C09109=1136.601,82.163,-54.023,-179.519,6.650,149.079
C09110=1136.606,81.914,-54.006,-179.522,6.649,149.080
C09111=1136.612,81.665,-53.989,-179.524,6.648,149.080
C09112=1136.617,81.416,-53.971,-179.527,6.646,149.081
C09113=1136.621,81.166,-53.954,-179.530,6.644,149.081
C09114=1136.626,80.916,-53.937,-179.532,6.643,149.082
C09115=1136.631,80.667,-53.920,-179.536,6.642,149.082
C09116=1136.636,80.418,-53.903,-179.538,6.641,149.083
C09117=1136.642,80.168,-53.886,-179.541,6.639,149.083
C09118=1136.646,79.919,-53.869,-179.543,6.637,149.084
C09119=1136.651,79.651,-53.850,-179.547,6.636,149.084
C09120=1136.656,79.383,-53.832,-179.549,6.634,149.085
C09121=1136.662,79.114,-53.813,-179.552,6.633,149.085
C09122=1136.668,78.846,-53.795,-179.555,6.632,149.086
C09123=1136.672,78.596,-53.778,-179.558,6.630,149.086
C09124=1136.677,78.347,-53.761,-179.560,6.629,149.087
C09125=1136.682,78.097,-53.744,-179.563,6.627,149.087
C09126=1136.687,77.847,-53.727,-179.566,6.626,149.088
C09127=1136.692,77.599,-53.710,-179.569,6.624,149.088
C09128=1136.697,77.349,-53.693,-179.571,6.624,149.089
C09129=1136.702,77.100,-53.676,-179.574,6.622,149.089
C09130=1136.706,76.850,-53.659,-179.577,6.621,149.090
C09131=1136.712,76.601,-53.642,-179.580,6.619,149.090
C09132=1136.716,76.352,-53.626,-179.582,6.618,149.091
C09133=1136.722,76.102,-53.609,-179.585,6.616,149.091
C09134=1136.727,75.853,-53.592,-179.587,6.615,149.091
C09135=1136.732,75.603,-53.575,-179.591,6.614,149.092
C09136=1136.736,75.354,-53.558,-179.593,6.613,149.093
C09137=1136.741,75.105,-53.540,-179.596,6.611,149.093
C09138=1136.746,74.856,-53.524,-179.598,6.609,149.093
C09139=1136.751,74.606,-53.507,-179.601,6.608,149.094
C09140=1136.756,74.357,-53.490,-179.604,6.607,149.095
C09141=1136.761,74.108,-53.474,-179.606,6.606,149.095
C09142=1136.766,73.858,-53.456,-179.609,6.604,149.095
C09143=1136.771,73.609,-53.440,-179.612,6.603,149.096
C09144=1136.775,73.359,-53.423,-179.615,6.602,149.096
C09145=1136.781,73.110,-53.406,-179.617,6.600,149.097
C09146=1136.786,72.860,-53.390,-179.620,6.598,149.097
C09147=1136.790,72.610,-53.374,-179.623,6.597,149.098
C09148=1136.796,72.361,-53.357,-179.625,6.596,149.098
C09149=1136.801,72.112,-53.340,-179.628,6.595,149.099
C09150=1136.806,71.863,-53.324,-179.631,6.593,149.099
C09151=1136.811,71.613,-53.307,-179.633,6.592,149.100
C09152=1136.816,71.364,-53.290,-179.636,6.591,149.100
C09153=1136.821,71.115,-53.274,-179.639,6.589,149.101
C09154=1136.826,70.865,-53.256,-179.642,6.588,149.101
C09155=1136.830,70.616,-53.240,-179.644,6.587,149.102
C09156=1136.836,70.366,-53.224,-179.647,6.585,149.102
C09157=1136.840,70.117,-53.207,-179.650,6.584,149.103
C09158=1136.845,69.867,-53.190,-179.652,6.583,149.103
C09159=1136.850,69.618,-53.174,-179.655,6.581,149.104
C09160=1136.855,69.369,-53.157,-179.658,6.580,149.104
C09161=1136.860,69.120,-53.141,-179.661,6.578,149.105
C09162=1136.866,68.870,-53.124,-179.663,6.578,149.105
C09163=1136.870,68.620,-53.108,-179.666,6.576,149.106
C09164=1136.875,68.371,-53.091,-179.669,6.575,149.106
C09165=1136.880,68.122,-53.075,-179.671,6.574,149.107
C09166=1136.886,67.872,-53.058,-179.674,6.572,149.107
C09167=1136.890,67.623,-53.042,-179.677,6.570,149.108
C09168=1136.895,67.374,-53.025,-179.679,6.570,149.108
C09169=1136.900,67.124,-53.009,-179.682,6.568,149.109
C09170=1136.905,66.874,-52.993,-179.685,6.567,149.109
C09171=1136.910,66.626,-52.977,-179.687,6.566,149.110
C09172=1136.915,66.376,-52.959,-179.690,6.565,149.110
C09173=1136.920,66.126,-52.944,-179.693,6.563,149.111
C09174=1136.925,65.877,-52.927,-179.695,6.562,149.111
C09175=1136.930,65.628,-52.911,-179.698,6.561,149.112
C09176=1136.935,65.378,-52.895,-179.701,6.559,149.112
C09177=1136.940,65.129,-52.878,-179.704,6.558,149.113
C09178=1136.944,64.880,-52.862,-179.706,6.557,149.113
C09179=1136.950,64.630,-52.846,-179.709,6.555,149.114
C09180=1136.955,64.380,-52.829,-179.712,6.554,149.114
C09181=1136.960,64.132,-52.813,-179.714,6.553,149.115
C09182=1136.965,63.882,-52.797,-179.717,6.551,149.115
C09183=1136.970,63.633,-52.780,-179.719,6.551,149.116
C09184=1136.974,63.383,-52.764,-179.722,6.549,149.116
C09185=1136.980,63.134,-52.748,-179.725,6.548,149.117
C09186=1136.984,62.884,-52.732,-179.728,6.547,149.117
C09187=1136.989,62.635,-52.716,-179.730,6.545,149.118
C09188=1136.994,62.385,-52.700,-179.733,6.544,149.118
C09189=1136.999,62.136,-52.684,-179.735,6.543,149.119
C09190=1137.004,61.886,-52.668,-179.738,6.542,149.119
C09191=1137.009,61.637,-52.651,-179.741,6.540,149.120
C09192=1137.015,61.387,-52.635,-179.743,6.539,149.120
C09193=1137.020,61.138,-52.618,-179.746,6.538,149.120
C09194=1137.025,60.888,-52.603,-179.749,6.536,149.121
C09195=1137.030,60.639,-52.586,-179.752,6.535,149.122
C09196=1137.034,60.389,-52.570,-179.754,6.534,149.122
C09197=1137.040,60.140,-52.554,-179.758,6.532,149.123
C09198=1137.045,59.891,-52.538,-179.760,6.532,149.123
C09199=1137.049,59.641,-52.522,-179.762,6.530,149.124
C09200=1137.055,59.392,-52.506,-179.765,6.529,149.124
C09201=1137.059,59.142,-52.491,-179.768,6.528,149.125
C09202=1137.064,58.893,-52.474,-179.771,6.526,149.125
C09203=1137.069,58.644,-52.459,-179.773,6.525,149.126
C09204=1137.074,58.395,-52.442,-179.776,6.524,149.126
C09205=1137.079,58.145,-52.427,-179.779,6.522,149.127
C09206=1137.084,57.895,-52.411,-179.781,6.522,149.127
C09207=1137.089,57.646,-52.394,-179.784,6.520,149.128
C09208=1137.094,57.397,-52.379,-179.786,6.520,149.128
C09209=1137.099,57.147,-52.363,-179.789,6.518,149.129
C09210=1137.104,56.898,-52.347,-179.792,6.516,149.129
C09211=1137.109,56.648,-52.331,-179.794,6.516,149.130
C09212=1137.114,56.398,-52.315,-179.797,6.514,149.130
C09213=1137.120,56.149,-52.299,-179.799,6.513,149.131
C09214=1137.124,55.900,-52.283,-179.802,6.512,149.131
C09215=1137.129,55.650,-52.268,-179.805,6.510,149.132
C09216=1137.134,55.401,-52.252,-179.807,6.510,149.132
C09217=1137.139,55.151,-52.236,-179.810,6.508,149.133
C09218=1137.144,54.902,-52.220,-179.813,6.507,149.133
C09219=1137.150,54.653,-52.204,-179.816,6.506,149.134
C09220=1137.154,54.403,-52.188,-179.818,6.504,149.134
C09221=1137.159,54.154,-52.173,-179.821,6.504,149.135
C09222=1137.164,53.904,-52.158,-179.824,6.502,149.135
C09223=1137.170,53.636,-52.141,-179.827,6.500,149.136
C09224=1137.175,53.367,-52.123,-179.829,6.500,149.136
C09225=1137.180,53.098,-52.106,-179.832,6.498,149.137
C09226=1137.186,52.830,-52.089,-179.835,6.497,149.138
C09227=1137.191,52.580,-52.074,-179.837,6.496,149.138
C09228=1137.196,52.331,-52.059,-179.840,6.495,149.138
C09229=1137.201,52.081,-52.043,-179.843,6.493,149.139
C09230=1137.206,51.832,-52.027,-179.845,6.492,149.140
C09231=1137.211,51.583,-52.011,-179.848,6.491,149.140
C09232=1137.215,51.333,-51.996,-179.851,6.490,149.141
C09233=1137.221,51.084,-51.980,-179.854,6.489,149.141
C09234=1137.226,50.834,-51.964,-179.856,6.488,149.142
C09235=1137.232,50.585,-51.949,-179.859,6.487,149.142
C09236=1137.236,50.335,-51.933,-179.862,6.485,149.143
C09237=1137.241,50.086,-51.918,-179.864,6.484,149.143
C09238=1137.246,49.836,-51.902,-179.867,6.483,149.144
C09239=1137.252,49.587,-51.887,-179.869,6.482,149.144
C09240=1137.256,49.337,-51.871,-179.872,6.480,149.145
C09241=1137.261,49.088,-51.856,-179.874,6.480,149.145
C09242=1137.267,48.838,-51.840,-179.878,6.478,149.146
C09243=1137.271,48.589,-51.825,-179.880,6.477,149.146
C09244=1137.276,48.339,-51.809,-179.882,6.476,149.147
C09245=1137.281,48.090,-51.794,-179.886,6.475,149.147
C09246=1137.286,47.840,-51.779,-179.888,6.474,149.148
C09247=1137.291,47.591,-51.763,-179.891,6.472,149.148
C09248=1137.297,47.342,-51.747,-179.893,6.472,149.149
C09249=1137.301,47.092,-51.732,-179.896,6.470,149.149
C09250=1137.306,46.842,-51.716,-179.898,6.469,149.150
C09251=1137.311,46.593,-51.701,-179.901,6.468,149.150
C09252=1137.317,46.343,-51.687,-179.904,6.467,149.151
C09253=1137.322,46.094,-51.671,-179.906,6.466,149.151
C09254=1137.326,45.844,-51.656,-179.908,6.465,149.152
C09255=1137.331,45.595,-51.640,-179.912,6.463,149.152
C09256=1137.336,45.346,-51.625,-179.914,6.463,149.153
C09257=1137.341,45.096,-51.609,-179.917,6.461,149.153
C09258=1137.347,44.847,-51.594,-179.920,6.460,149.154
C09259=1137.352,44.597,-51.580,-179.922,6.459,149.154
C09260=1137.357,44.347,-51.564,-179.925,6.457,149.155
C09261=1137.361,44.098,-51.549,-179.927,6.457,149.156
C09262=1137.367,43.849,-51.533,-179.930,6.455,149.156
C09263=1137.371,43.599,-51.518,-179.932,6.454,149.156
C09264=1137.377,43.349,-51.503,-179.936,6.453,149.157
C09265=1137.382,43.100,-51.488,-179.938,6.452,149.158
C09266=1137.387,42.851,-51.473,-179.941,6.451,149.158
C09267=1137.392,42.602,-51.458,-179.943,6.450,149.159
C09268=1137.397,42.351,-51.442,-179.946,6.449,149.159
C09269=1137.401,42.102,-51.427,-179.948,6.448,149.160
C09270=1137.407,41.853,-51.412,-179.951,6.446,149.160
C09271=1137.411,41.604,-51.397,-179.954,6.446,149.161
C09272=1137.417,41.354,-51.382,-179.956,6.444,149.161
C09273=1137.422,41.104,-51.367,-179.959,6.444,149.162
C09274=1137.427,40.855,-51.351,-179.962,6.442,149.162
C09275=1137.432,40.605,-51.337,-179.964,6.441,149.163
C09276=1137.437,40.356,-51.322,-179.967,6.440,149.163
C09277=1137.442,40.107,-51.307,-179.969,6.439,149.164
C09278=1137.448,39.857,-51.292,-179.972,6.437,149.164
C09279=1137.452,39.608,-51.277,-179.975,6.437,149.165
C09280=1137.457,39.358,-51.261,-179.977,6.435,149.165
C09281=1137.462,39.108,-51.246,-179.980,6.434,149.166
C09282=1137.467,38.859,-51.231,-179.983,6.433,149.167
C09283=1137.473,38.609,-51.217,-179.985,6.432,149.167
C09284=1137.477,38.360,-51.202,-179.987,6.432,149.167
C09285=1137.483,38.110,-51.186,-179.990,6.430,149.168
C09286=1137.488,37.861,-51.172,-179.993,6.429,149.169
C09287=1137.493,37.611,-51.156,-179.995,6.428,149.169
C09288=1137.498,37.361,-51.142,-179.998,6.427,149.170
C09289=1137.503,37.112,-51.127,179.999,6.426,149.170
C09290=1137.508,36.862,-51.112,179.997,6.425,149.171
C09291=1137.513,36.613,-51.097,179.994,6.424,149.171
C09292=1137.518,36.364,-51.083,179.992,6.423,149.172
C09293=1137.523,36.114,-51.067,179.989,6.421,149.172
C09294=1137.528,35.864,-51.053,179.986,6.421,149.173
C09295=1137.533,35.615,-51.038,179.984,6.419,149.173
C09296=1137.539,35.365,-51.023,179.981,6.418,149.174
C09297=1137.543,35.116,-51.008,179.978,6.417,149.174
C09298=1137.548,34.867,-50.994,179.976,6.416,149.175
C09299=1137.554,34.617,-50.978,179.974,6.415,149.175
C09300=1137.558,34.367,-50.964,179.971,6.414,149.176
C09301=1137.563,34.118,-50.949,179.968,6.413,149.176
C09302=1137.569,33.868,-50.934,179.966,6.412,149.177
C09303=1137.574,33.619,-50.920,179.963,6.411,149.178
C09304=1137.578,33.370,-50.905,179.960,6.410,149.178
C09305=1137.584,33.121,-50.891,179.958,6.409,149.178
C09306=1137.589,32.871,-50.875,179.955,6.408,149.179
C09307=1137.594,32.621,-50.861,179.953,6.407,149.180
C09308=1137.599,32.372,-50.847,179.950,6.406,149.180
C09309=1137.604,32.123,-50.832,179.947,6.405,149.181
C09310=1137.610,31.873,-50.817,179.945,6.404,149.181
C09311=1137.615,31.623,-50.803,179.942,6.403,149.182
C09312=1137.619,31.374,-50.788,179.940,6.402,149.182
C09313=1137.624,31.124,-50.773,179.937,6.400,149.183
C09314=1137.630,30.874,-50.758,179.934,6.400,149.183
C09315=1137.635,30.625,-50.743,179.932,6.399,149.184
C09316=1137.639,30.375,-50.729,179.929,6.397,149.184
C09317=1137.644,30.126,-50.715,179.927,6.397,149.185
C09318=1137.650,29.877,-50.701,179.924,6.395,149.185
C09319=1137.655,29.627,-50.686,179.922,6.394,149.186
C09320=1137.660,29.377,-50.671,179.919,6.394,149.187
C09321=1137.665,29.128,-50.657,179.916,6.392,149.187
C09322=1137.670,28.878,-50.642,179.914,6.391,149.188
C09323=1137.675,28.629,-50.628,179.911,6.390,149.188
C09324=1137.680,28.379,-50.613,179.909,6.389,149.189
C09325=1137.685,28.129,-50.599,179.907,6.389,149.189
C09326=1137.691,27.880,-50.584,179.903,6.387,149.190
C09327=1137.696,27.611,-50.569,179.901,6.387,149.190
C09328=1137.701,27.343,-50.553,179.898,6.385,149.191
C09329=1137.707,27.073,-50.538,179.895,6.384,149.191
C09330=1137.712,26.804,-50.522,179.892,6.383,149.192
C09331=1137.718,26.554,-50.507,179.890,6.382,149.193
C09332=1137.723,26.305,-50.493,179.887,6.381,149.193
C09333=1137.728,26.056,-50.479,179.885,6.380,149.194
C09334=1137.733,25.806,-50.465,179.882,6.379,149.194
C09335=1137.738,25.556,-50.451,179.879,6.378,149.195
C09336=1137.743,25.307,-50.436,179.877,6.377,149.195
C09337=1137.748,25.057,-50.421,179.875,6.376,149.196
C09338=1137.753,24.808,-50.408,179.872,6.375,149.196
C09339=1137.758,24.559,-50.393,179.869,6.374,149.197
C09340=1137.763,24.309,-50.379,179.867,6.373,149.197
C09341=1137.768,24.059,-50.365,179.864,6.373,149.198
C09342=1137.773,23.810,-50.350,179.862,6.371,149.198
C09343=1137.779,23.561,-50.337,179.859,6.370,149.199
C09344=1137.783,23.311,-50.322,179.856,6.369,149.200
C09345=1137.788,23.061,-50.308,179.854,6.368,149.200
C09346=1137.793,22.811,-50.294,179.851,6.368,149.201
C09347=1137.798,22.562,-50.279,179.849,6.366,149.201
C09348=1137.804,22.313,-50.265,179.846,6.365,149.202
C09349=1137.809,22.063,-50.251,179.844,6.365,149.202
C09350=1137.814,21.813,-50.237,179.841,6.363,149.203
C09351=1137.819,21.564,-50.223,179.839,6.362,149.203
C09352=1137.824,21.315,-50.209,179.836,6.362,149.204
C09353=1137.829,21.065,-50.194,179.833,6.360,149.204
C09354=1137.834,20.815,-50.180,179.831,6.359,149.205
C09355=1137.839,20.565,-50.166,179.828,6.358,149.205
C09356=1137.845,20.316,-50.152,179.826,6.357,149.206
C09357=1137.850,20.067,-50.138,179.823,6.357,149.207
C09358=1137.855,19.816,-50.124,179.820,6.355,149.207
C09359=1137.861,19.567,-50.110,179.818,6.354,149.208
C09360=1137.865,19.318,-50.097,179.816,6.354,149.208
C09361=1137.870,19.068,-50.082,179.813,6.352,149.209
C09362=1137.875,18.819,-50.068,179.811,6.352,149.209
C09363=1137.880,18.570,-50.054,179.808,6.351,149.210
C09364=1137.885,18.320,-50.040,179.805,6.350,149.210
C09365=1137.890,18.069,-50.026,179.803,6.349,149.211
C09366=1137.896,17.820,-50.012,179.800,6.348,149.211
C09367=1137.901,17.571,-49.998,179.798,6.347,149.212
C09368=1137.906,17.321,-49.984,179.795,6.346,149.213
C09369=1137.911,17.072,-49.970,179.793,6.345,149.213
C09370=1137.916,16.823,-49.956,179.790,6.344,149.213
C09371=1137.921,16.572,-49.943,179.787,6.343,149.214
C09372=1137.926,16.323,-49.929,179.785,6.343,149.215
C09373=1137.931,16.074,-49.914,179.782,6.341,149.215
C09374=1137.936,15.824,-49.900,179.780,6.341,149.216
C09375=1137.942,15.575,-49.888,179.778,6.340,149.216
C09376=1137.946,15.325,-49.873,179.775,6.338,149.217
C09377=1137.951,15.075,-49.859,179.772,6.338,149.217
C09378=1137.957,14.826,-49.845,179.770,6.337,149.218
C09379=1137.962,14.576,-49.832,179.767,6.336,149.219
C09380=1137.967,14.327,-49.818,179.765,6.335,149.219
C09381=1137.972,14.077,-49.804,179.762,6.334,149.219
C09382=1137.977,13.827,-49.790,179.760,6.334,149.220
C09383=1137.983,13.578,-49.776,179.757,6.332,149.221
C09384=1137.987,13.329,-49.763,179.755,6.331,149.221
C09385=1137.992,13.078,-49.749,179.752,6.331,149.222
C09386=1137.998,12.829,-49.735,179.749,6.329,149.222
C09387=1138.003,12.580,-49.721,179.747,6.328,149.223
C09388=1138.008,12.330,-49.708,179.744,6.328,149.223
C09389=1138.013,12.081,-49.694,179.742,6.327,149.224
C09390=1138.019,11.831,-49.681,179.739,6.326,149.224
C09391=1138.024,11.581,-49.667,179.737,6.325,149.225
C09392=1138.028,11.332,-49.653,179.735,6.324,149.225
C09393=1138.034,11.082,-49.640,179.731,6.323,149.226
C09394=1138.039,10.833,-49.626,179.729,6.322,149.227
C09395=1138.044,10.583,-49.613,179.727,6.321,149.227
C09396=1138.049,10.333,-49.599,179.724,6.321,149.228
C09397=1138.055,10.084,-49.585,179.722,6.319,149.228
C09398=1138.059,9.834,-49.572,179.719,6.319,149.229
C09399=1138.064,9.585,-49.558,179.717,6.318,149.229
C09400=1138.070,9.335,-49.544,179.714,6.316,149.230
C09401=1138.074,9.086,-49.531,179.711,6.316,149.230
C09402=1138.080,8.836,-49.517,179.709,6.315,149.231
C09403=1138.085,8.586,-49.503,179.707,6.314,149.231
C09404=1138.090,8.337,-49.491,179.704,6.313,149.232
C09405=1138.095,8.087,-49.476,179.702,6.312,149.233
C09406=1138.101,7.838,-49.463,179.699,6.312,149.233
C09407=1138.105,7.588,-49.450,179.697,6.311,149.234
C09408=1138.111,7.339,-49.436,179.694,6.310,149.234
C09409=1138.115,7.089,-49.423,179.691,6.309,149.235
C09410=1138.121,6.840,-49.409,179.689,6.308,149.235
C09411=1138.126,6.589,-49.396,179.686,6.307,149.236
C09412=1138.131,6.341,-49.382,179.684,6.306,149.236
C09413=1138.136,6.090,-49.369,179.682,6.305,149.237
C09414=1138.141,5.841,-49.356,179.679,6.305,149.237
C09415=1138.146,5.591,-49.342,179.676,6.303,149.238
C09416=1138.151,5.342,-49.329,179.674,6.303,149.238
C09417=1138.156,5.092,-49.315,179.671,6.302,149.239
C09418=1138.161,4.843,-49.303,179.669,6.301,149.240
C09419=1138.167,4.593,-49.289,179.666,6.300,149.240
C09420=1138.172,4.344,-49.275,179.664,6.299,149.241
C09421=1138.177,4.094,-49.262,179.662,6.299,149.241
C09422=1138.183,3.844,-49.249,179.659,6.298,149.242
C09423=1138.187,3.595,-49.236,179.657,6.297,149.242
C09424=1138.193,3.345,-49.222,179.654,6.296,149.243
C09425=1138.198,3.096,-49.209,179.651,6.295,149.244
C09426=1138.203,2.846,-49.195,179.649,6.294,149.244
C09427=1138.208,2.597,-49.183,179.647,6.294,149.244
C09428=1138.213,2.346,-49.169,179.644,6.292,149.245
C09429=1138.218,2.097,-49.156,179.642,6.292,149.246
C09430=1138.224,1.848,-49.142,179.639,6.291,149.246
C09431=1138.229,1.578,-49.129,179.637,6.290,149.247
C09432=1138.235,1.308,-49.115,179.634,6.289,149.247
C09433=1138.240,1.039,-49.100,179.631,6.288,149.248
C09434=1138.246,0.770,-49.086,179.628,6.287,149.249
C09435=1138.251,0.519,-49.073,179.626,6.286,149.249
C09436=1138.256,0.271,-49.059,179.624,6.286,149.250
C09437=1138.261,0.021,-49.047,179.621,6.285,149.250
C09438=1138.266,-0.229,-49.033,179.618,6.283,149.251
C09439=1138.271,-0.478,-49.021,179.616,6.283,149.251
C09440=1138.277,-0.729,-49.007,179.613,6.282,149.252
C09441=1138.281,-0.977,-48.994,179.611,6.281,149.252
C09442=1138.287,-1.227,-48.981,179.609,6.281,149.253
C09443=1138.292,-1.477,-48.968,179.606,6.279,149.254
C09444=1138.297,-1.726,-48.955,179.604,6.279,149.254
C09445=1138.303,-1.976,-48.942,179.601,6.278,149.255
C09446=1138.307,-2.226,-48.929,179.599,6.277,149.255
C09447=1138.312,-2.475,-48.916,179.597,6.277,149.256
C09448=1138.318,-2.725,-48.903,179.593,6.275,149.256
C09449=1138.323,-2.975,-48.890,179.591,6.275,149.257
C09450=1138.328,-3.224,-48.876,179.589,6.274,149.257
C09451=1138.333,-3.473,-48.863,179.586,6.273,149.258
C09452=1138.338,-3.723,-48.851,179.584,6.273,149.258
C09453=1138.344,-3.973,-48.837,179.581,6.271,149.259
C09454=1138.349,-4.222,-48.825,179.579,6.271,149.260
C09455=1138.353,-4.472,-48.812,179.577,6.270,149.260
C09456=1138.359,-4.722,-48.799,179.574,6.269,149.261
C09457=1138.364,-4.971,-48.786,179.572,6.269,149.261
C09458=1138.369,-5.221,-48.773,179.570,6.268,149.262
C09459=1138.374,-5.470,-48.760,179.566,6.267,149.262
C09460=1138.380,-5.720,-48.747,179.564,6.266,149.263
C09461=1138.385,-5.969,-48.735,179.561,6.265,149.263
C09462=1138.390,-6.219,-48.722,179.559,6.264,149.264
C09463=1138.395,-6.469,-48.708,179.557,6.264,149.264
C09464=1138.401,-6.718,-48.696,179.554,6.263,149.265
C09465=1138.405,-6.968,-48.683,179.552,6.262,149.266
C09466=1138.410,-7.218,-48.670,179.549,6.261,149.266
C09467=1138.416,-7.467,-48.657,179.547,6.260,149.267
C09468=1138.421,-7.717,-48.644,179.545,6.260,149.267
C09469=1138.426,-7.967,-48.632,179.542,6.259,149.268
C09470=1138.431,-8.217,-48.620,179.540,6.258,149.268
C09471=1138.436,-8.466,-48.607,179.537,6.257,149.269
C09472=1138.442,-8.716,-48.594,179.534,6.256,149.270
C09473=1138.447,-8.966,-48.581,179.532,6.256,149.270
C09474=1138.452,-9.215,-48.568,179.530,6.255,149.270
C09475=1138.457,-9.464,-48.556,179.527,6.254,149.271
C09476=1138.462,-9.714,-48.543,179.525,6.254,149.272
C09477=1138.467,-9.964,-48.530,179.522,6.252,149.272
C09478=1138.473,-10.214,-48.518,179.520,6.252,149.273
C09479=1138.478,-10.463,-48.505,179.518,6.251,149.273
C09480=1138.483,-10.712,-48.492,179.515,6.250,149.274
C09481=1138.488,-10.962,-48.480,179.513,6.250,149.274
C09482=1138.493,-11.212,-48.467,179.511,6.249,149.275
C09483=1138.498,-11.461,-48.454,179.508,6.248,149.276
C09484=1138.504,-11.711,-48.442,179.506,6.248,149.276
C09485=1138.509,-11.961,-48.429,179.503,6.246,149.276
C09486=1138.514,-12.210,-48.417,179.500,6.246,149.277
C09487=1138.519,-12.460,-48.404,179.498,6.245,149.278
C09488=1138.524,-12.710,-48.392,179.495,6.244,149.278
C09489=1138.529,-12.959,-48.379,179.493,6.244,149.279
C09490=1138.534,-13.209,-48.367,179.491,6.243,149.279
C09491=1138.540,-13.458,-48.353,179.488,6.242,149.280
C09492=1138.545,-13.709,-48.341,179.486,6.241,149.280
C09493=1138.550,-13.958,-48.328,179.483,6.240,149.281
C09494=1138.555,-14.207,-48.316,179.481,6.240,149.282
C09495=1138.560,-14.457,-48.303,179.479,6.239,149.282
C09496=1138.566,-14.707,-48.291,179.476,6.238,149.283
C09497=1138.571,-14.956,-48.279,179.474,6.238,149.283
C09498=1138.576,-15.205,-48.266,179.472,6.237,149.284
C09499=1138.581,-15.456,-48.254,179.469,6.236,149.284
C09500=1138.586,-15.705,-48.241,179.467,6.236,149.285
C09501=1138.591,-15.955,-48.229,179.464,6.234,149.285
C09502=1138.597,-16.205,-48.217,179.461,6.234,149.286
C09503=1138.602,-16.454,-48.204,179.459,6.233,149.287
C09504=1138.607,-16.703,-48.192,179.457,6.232,149.287
C09505=1138.612,-16.953,-48.180,179.454,6.232,149.288
C09506=1138.617,-17.202,-48.167,179.452,6.231,149.288
C09507=1138.622,-17.453,-48.155,179.449,6.230,149.289
C09508=1138.627,-17.702,-48.142,179.447,6.230,149.289
C09509=1138.632,-17.952,-48.130,179.445,6.229,149.290
C09510=1138.638,-18.202,-48.118,179.442,6.228,149.290
C09511=1138.643,-18.451,-48.105,179.440,6.227,149.291
C09512=1138.648,-18.701,-48.093,179.437,6.226,149.291
C09513=1138.654,-18.950,-48.081,179.435,6.226,149.292
C09514=1138.659,-19.200,-48.069,179.433,6.225,149.293
C09515=1138.664,-19.449,-48.056,179.430,6.224,149.293
C09516=1138.670,-19.699,-48.044,179.428,6.224,149.294
C09517=1138.675,-19.949,-48.032,179.426,6.223,149.294
C09518=1138.680,-20.199,-48.020,179.423,6.222,149.295
C09519=1138.685,-20.449,-48.007,179.421,6.222,149.295
C09520=1138.690,-20.699,-47.995,179.419,6.221,149.296
C09521=1138.695,-20.948,-47.982,179.416,6.220,149.297
C09522=1138.701,-21.198,-47.971,179.413,6.219,149.297
C09523=1138.706,-21.447,-47.958,179.411,6.218,149.298
C09524=1138.711,-21.697,-47.946,179.408,6.218,149.298
C09525=1138.716,-21.946,-47.933,179.406,6.217,149.299
C09526=1138.722,-22.196,-47.922,179.404,6.216,149.299
C09527=1138.726,-22.445,-47.910,179.401,6.216,149.300
C09528=1138.732,-22.695,-47.898,179.399,6.215,149.300
C09529=1138.737,-22.945,-47.885,179.397,6.214,149.301
C09530=1138.742,-23.195,-47.873,179.394,6.214,149.301
C09531=1138.748,-23.445,-47.861,179.392,6.213,149.302
C09532=1138.753,-23.694,-47.849,179.389,6.212,149.303
C09533=1138.758,-23.944,-47.837,179.387,6.212,149.303
C09534=1138.763,-24.193,-47.824,179.385,6.211,149.304
C09535=1138.769,-24.463,-47.812,179.382,6.210,149.304
C09536=1138.774,-24.733,-47.799,179.379,6.209,149.305
C09537=1138.780,-25.003,-47.786,179.377,6.208,149.305
C09538=1138.786,-25.273,-47.773,179.375,6.208,149.306
C09539=1138.791,-25.523,-47.761,179.372,6.207,149.307
C09540=1138.796,-25.772,-47.749,179.370,6.206,149.307
C09541=1138.802,-26.022,-47.737,179.368,6.206,149.308
C09542=1138.807,-26.272,-47.725,179.365,6.205,149.308
C09543=1138.811,-26.521,-47.713,179.363,6.204,149.309
C09544=1138.817,-26.771,-47.701,179.360,6.204,149.309
C09545=1138.822,-27.021,-47.689,179.357,6.202,149.310
C09546=1138.827,-27.270,-47.676,179.355,6.202,149.310
C09547=1138.832,-27.520,-47.665,179.352,6.201,149.311
C09548=1138.838,-27.770,-47.653,179.350,6.200,149.312
C09549=1138.843,-28.020,-47.641,179.348,6.200,149.312
C09550=1138.848,-28.269,-47.629,179.345,6.199,149.313
C09551=1138.853,-28.519,-47.617,179.343,6.198,149.313
C09552=1138.858,-28.769,-47.606,179.341,6.198,149.314
C09553=1138.864,-29.019,-47.594,179.338,6.197,149.314
C09554=1138.869,-29.268,-47.581,179.336,6.197,149.315
C09555=1138.873,-29.518,-47.570,179.334,6.196,149.315
C09556=1138.880,-29.767,-47.558,179.331,6.195,149.316
C09557=1138.885,-30.017,-47.546,179.329,6.195,149.316
C09558=1138.890,-30.267,-47.535,179.327,6.194,149.317
C09559=1138.895,-30.516,-47.523,179.324,6.193,149.318
C09560=1138.900,-30.766,-47.511,179.322,6.193,149.318
C09561=1138.906,-31.016,-47.499,179.319,6.192,149.319
C09562=1138.910,-31.265,-47.487,179.317,6.191,149.319
C09563=1138.916,-31.515,-47.476,179.315,6.191,149.320
C09564=1138.921,-31.765,-47.464,179.312,6.190,149.320
C09565=1138.926,-32.015,-47.452,179.310,6.189,149.321
C09566=1138.932,-32.263,-47.440,179.308,6.189,149.321
C09567=1138.937,-32.513,-47.428,179.305,6.188,149.322
C09568=1138.942,-32.763,-47.417,179.303,6.187,149.323
C09569=1138.947,-33.013,-47.405,179.301,6.187,149.323
C09570=1138.953,-33.263,-47.393,179.298,6.186,149.324
C09571=1138.957,-33.512,-47.382,179.296,6.185,149.324
C09572=1138.963,-33.762,-47.370,179.294,6.185,149.325
C09573=1138.969,-34.012,-47.359,179.291,6.184,149.325
C09574=1138.973,-34.261,-47.347,179.289,6.183,149.326
C09575=1138.979,-34.511,-47.335,179.287,6.183,149.326
C09576=1138.984,-34.761,-47.324,179.284,6.182,149.327
C09577=1138.989,-35.011,-47.312,179.282,6.182,149.328
C09578=1138.994,-35.261,-47.300,179.280,6.181,149.328
C09579=1139.000,-35.510,-47.289,179.277,6.180,149.329
C09580=1139.005,-35.760,-47.278,179.275,6.180,149.329
C09581=1139.010,-36.009,-47.266,179.273,6.179,149.330
C09582=1139.015,-36.259,-47.254,179.270,6.178,149.330
C09583=1139.021,-36.509,-47.242,179.268,6.178,149.331
C09584=1139.026,-36.758,-47.232,179.266,6.177,149.331
C09585=1139.031,-37.008,-47.220,179.263,6.176,149.332
C09586=1139.036,-37.258,-47.208,179.261,6.176,149.333
C09587=1139.041,-37.508,-47.196,179.259,6.175,149.333
C09588=1139.046,-37.757,-47.185,179.256,6.174,149.334
C09589=1139.052,-38.006,-47.174,179.254,6.174,149.334
C09590=1139.057,-38.256,-47.162,179.252,6.173,149.335
C09591=1139.062,-38.506,-47.150,179.249,6.172,149.335
C09592=1139.067,-38.756,-47.139,179.247,6.172,149.336
C09593=1139.072,-39.005,-47.127,179.245,6.171,149.336
C09594=1139.078,-39.254,-47.116,179.242,6.171,149.337
C09595=1139.083,-39.504,-47.104,179.240,6.170,149.337
C09596=1139.089,-39.755,-47.093,179.238,6.169,149.338
C09597=1139.094,-40.005,-47.082,179.236,6.169,149.339
C09598=1139.100,-40.254,-47.071,179.233,6.169,149.339
C09599=1139.104,-40.503,-47.059,179.231,6.168,149.340
C09600=1139.109,-40.753,-47.048,179.229,6.167,149.340
C09601=1139.114,-41.003,-47.036,179.226,6.167,149.341
C09602=1139.120,-41.252,-47.025,179.224,6.166,149.341
C09603=1139.125,-41.502,-47.014,179.222,6.165,149.342
C09604=1139.130,-41.752,-47.003,179.219,6.165,149.342
C09605=1139.136,-42.001,-46.991,179.217,6.164,149.343
C09606=1139.141,-42.251,-46.980,179.215,6.163,149.344
C09607=1139.146,-42.501,-46.968,179.212,6.163,149.344
C09608=1139.151,-42.750,-46.957,179.210,6.162,149.345
C09609=1139.157,-43.000,-46.946,179.207,6.162,149.345
C09610=1139.162,-43.250,-46.935,179.205,6.161,149.346
C09611=1139.167,-43.500,-46.923,179.203,6.160,149.346
C09612=1139.173,-43.749,-46.912,179.200,6.160,149.347
C09613=1139.178,-43.999,-46.901,179.198,6.159,149.347
C09614=1139.183,-44.249,-46.889,179.196,6.158,149.348
C09615=1139.188,-44.499,-46.878,179.193,6.158,149.349
C09616=1139.193,-44.748,-46.867,179.192,6.158,149.349
C09617=1139.199,-44.998,-46.856,179.190,6.157,149.350
C09618=1139.204,-45.248,-46.845,179.187,6.156,149.350
C09619=1139.209,-45.497,-46.834,179.185,6.156,149.351
C09620=1139.215,-45.747,-46.823,179.183,6.155,149.351
C09621=1139.219,-45.997,-46.811,179.180,6.155,149.352
C09622=1139.225,-46.246,-46.800,179.178,6.154,149.352
C09623=1139.230,-46.496,-46.789,179.176,6.153,149.353
C09624=1139.235,-46.746,-46.778,179.173,6.153,149.354
C09625=1139.241,-46.995,-46.766,179.171,6.152,149.354
C09626=1139.246,-47.245,-46.756,179.168,6.151,149.354
C09627=1139.251,-47.495,-46.744,179.166,6.151,149.355
C09628=1139.257,-47.744,-46.733,179.164,6.150,149.356
C09629=1139.262,-47.995,-46.722,179.162,6.150,149.356
C09630=1139.267,-48.243,-46.711,179.160,6.149,149.357
C09631=1139.273,-48.493,-46.700,179.157,6.149,149.357
C09632=1139.278,-48.744,-46.689,179.155,6.148,149.358
C09633=1139.283,-48.993,-46.678,179.153,6.147,149.358
C09634=1139.288,-49.243,-46.668,179.150,6.147,149.359
C09635=1139.293,-49.493,-46.656,179.148,6.146,149.359
C09636=1139.299,-49.742,-46.645,179.146,6.145,149.360
C09637=1139.304,-49.992,-46.634,179.143,6.145,149.361
C09638=1139.310,-50.241,-46.623,179.141,6.144,149.361
C09639=1139.314,-50.512,-46.611,179.139,6.143,149.362
C09640=1139.320,-50.783,-46.599,179.136,6.143,149.362
C09641=1139.327,-51.054,-46.588,179.134,6.142,149.363
C09642=1139.332,-51.325,-46.575,179.131,6.142,149.364
C09643=1139.337,-51.574,-46.564,179.129,6.141,149.364
C09644=1139.342,-51.824,-46.554,179.126,6.141,149.365
C09645=1139.347,-52.073,-46.542,179.124,6.140,149.365
C09646=1139.354,-52.323,-46.532,179.123,6.140,149.366
C09647=1139.358,-52.573,-46.520,179.120,6.139,149.366
C09648=1139.364,-52.822,-46.510,179.118,6.139,149.367
C09649=1139.368,-53.072,-46.499,179.116,6.138,149.367
C09650=1139.373,-53.322,-46.488,179.113,6.137,149.368
C09651=1139.380,-53.572,-46.477,179.111,6.137,149.368
C09652=1139.385,-53.822,-46.466,179.108,6.136,149.369
C09653=1139.390,-54.071,-46.455,179.106,6.135,149.369
C09654=1139.395,-54.321,-46.445,179.104,6.136,149.370
C09655=1139.400,-54.571,-46.435,179.102,6.135,149.371
C09656=1139.405,-54.820,-46.423,179.100,6.134,149.371
C09657=1139.411,-55.070,-46.412,179.097,6.134,149.372
C09658=1139.416,-55.320,-46.401,179.095,6.133,149.372
C09659=1139.422,-55.569,-46.391,179.093,6.132,149.373
C09660=1139.427,-55.819,-46.380,179.091,6.131,149.373
C09661=1139.431,-56.069,-46.369,179.088,6.131,149.374
C09662=1139.437,-56.319,-46.359,179.086,6.131,149.374
C09663=1139.442,-56.568,-46.348,179.084,6.130,149.375
C09664=1139.447,-56.818,-46.337,179.081,6.130,149.376
C09665=1139.453,-57.068,-46.326,179.079,6.129,149.376
C09666=1139.458,-57.317,-46.315,179.077,6.128,149.377
C09667=1139.463,-57.568,-46.305,179.075,6.127,149.377
C09668=1139.469,-57.817,-46.294,179.072,6.127,149.378
C09669=1139.474,-58.067,-46.283,179.071,6.127,149.378
C09670=1139.479,-58.316,-46.273,179.068,6.126,149.379
C09671=1139.484,-58.566,-46.262,179.066,6.126,149.379
C09672=1139.489,-58.815,-46.251,179.064,6.125,149.380
C09673=1139.494,-59.066,-46.241,179.061,6.124,149.380
C09674=1139.500,-59.315,-46.231,179.059,6.124,149.381
C09675=1139.505,-59.565,-46.219,179.057,6.123,149.382
C09676=1139.510,-59.814,-46.209,179.055,6.123,149.382
C09677=1139.517,-60.064,-46.198,179.053,6.122,149.383
C09678=1139.522,-60.314,-46.188,179.050,6.122,149.383
C09679=1139.527,-60.563,-46.177,179.048,6.121,149.384
C09680=1139.532,-60.814,-46.166,179.046,6.121,149.384
C09681=1139.538,-61.063,-46.156,179.044,6.120,149.385
C09682=1139.543,-61.313,-46.146,179.041,6.120,149.385
C09683=1139.548,-61.562,-46.135,179.039,6.119,149.386
C09684=1139.553,-61.813,-46.124,179.037,6.119,149.386
C09685=1139.558,-62.062,-46.114,179.034,6.118,149.387
C09686=1139.563,-62.312,-46.103,179.032,6.118,149.388
C09687=1139.569,-62.562,-46.093,179.030,6.117,149.388
C09688=1139.574,-62.811,-46.082,179.028,6.117,149.388
C09689=1139.579,-63.061,-46.072,179.026,6.116,149.389
C09690=1139.585,-63.311,-46.061,179.024,6.116,149.390
C09691=1139.590,-63.561,-46.051,179.021,6.115,149.390
C09692=1139.596,-63.810,-46.041,179.019,6.114,149.391
C09693=1139.601,-64.060,-46.030,179.017,6.114,149.391
C09694=1139.606,-64.310,-46.019,179.015,6.114,149.392
C09695=1139.611,-64.559,-46.009,179.013,6.113,149.392
C09696=1139.616,-64.809,-45.999,179.010,6.113,149.393
C09697=1139.621,-65.059,-45.989,179.008,6.112,149.393
C09698=1139.627,-65.308,-45.978,179.006,6.111,149.394
C09699=1139.632,-65.558,-45.968,179.003,6.110,149.394
C09700=1139.638,-65.808,-45.958,179.001,6.111,149.395
C09701=1139.643,-66.058,-45.947,178.999,6.110,149.396
C09702=1139.648,-66.308,-45.937,178.997,6.109,149.396
C09703=1139.653,-66.557,-45.926,178.995,6.108,149.397
C09704=1139.658,-66.807,-45.915,178.992,6.108,149.397
C09705=1139.664,-67.056,-45.905,178.991,6.108,149.398
C09706=1139.670,-67.306,-45.895,178.988,6.107,149.398
C09707=1139.675,-67.556,-45.884,178.986,6.107,149.399
C09708=1139.680,-67.806,-45.874,178.984,6.106,149.399
C09709=1139.685,-68.055,-45.865,178.981,6.105,149.400
C09710=1139.690,-68.305,-45.854,178.980,6.105,149.400
C09711=1139.696,-68.555,-45.844,178.977,6.105,149.401
C09712=1139.701,-68.804,-45.834,178.975,6.104,149.402
C09713=1139.706,-69.055,-45.823,178.973,6.103,149.402
C09714=1139.712,-69.304,-45.813,178.970,6.103,149.403
C09715=1139.717,-69.554,-45.803,178.968,6.103,149.403
C09716=1139.722,-69.804,-45.792,178.966,6.102,149.404
C09717=1139.727,-70.053,-45.782,178.964,6.102,149.404
C09718=1139.733,-70.303,-45.772,178.962,6.101,149.405
C09719=1139.738,-70.553,-45.762,178.959,6.100,149.405
C09720=1139.743,-70.802,-45.751,178.958,6.100,149.406
C09721=1139.749,-71.052,-45.741,178.955,6.100,149.406
C09722=1139.754,-71.302,-45.731,178.953,6.099,149.407
C09723=1139.759,-71.551,-45.721,178.951,6.099,149.408
C09724=1139.765,-71.801,-45.711,178.949,6.099,149.408
C09725=1139.770,-72.052,-45.701,178.947,6.098,149.409
C09726=1139.775,-72.301,-45.691,178.945,6.097,149.409
C09727=1139.781,-72.551,-45.681,178.942,6.097,149.410
C09728=1139.786,-72.800,-45.671,178.940,6.096,149.410
C09729=1139.791,-73.050,-45.660,178.938,6.096,149.411
C09730=1139.797,-73.300,-45.650,178.936,6.095,149.411
C09731=1139.802,-73.550,-45.640,178.933,6.095,149.412
C09732=1139.808,-73.799,-45.630,178.931,6.094,149.412
C09733=1139.812,-74.049,-45.620,178.929,6.094,149.413
C09734=1139.818,-74.299,-45.610,178.927,6.093,149.413
C09735=1139.823,-74.549,-45.600,178.925,6.093,149.414
C09736=1139.829,-74.798,-45.590,178.922,6.092,149.415
C09737=1139.833,-75.048,-45.580,178.921,6.092,149.415
C09738=1139.839,-75.298,-45.570,178.919,6.091,149.415
C09739=1139.845,-75.547,-45.559,178.916,6.091,149.416
C09740=1139.850,-75.797,-45.550,178.914,6.090,149.417
C09741=1139.855,-76.047,-45.540,178.912,6.090,149.417
C09742=1139.860,-76.297,-45.530,178.910,6.090,149.418
C09743=1139.866,-76.569,-45.518,178.907,6.089,149.418
C09744=1139.872,-76.840,-45.508,178.905,6.088,149.419
C09745=1139.877,-77.111,-45.497,178.903,6.088,149.419
C09746=1139.883,-77.383,-45.486,178.900,6.087,149.420
C09747=1139.889,-77.633,-45.476,178.898,6.087,149.421
C09748=1139.894,-77.882,-45.467,178.896,6.087,149.421
C09749=1139.900,-78.132,-45.457,178.894,6.086,149.422
C09750=1139.905,-78.381,-45.446,178.892,6.085,149.422
C09751=1139.910,-78.632,-45.437,178.889,6.085,149.423
C09752=1139.916,-78.881,-45.427,178.888,6.085,149.423
C09753=1139.921,-79.131,-45.417,178.886,6.084,149.424
C09754=1139.926,-79.381,-45.408,178.883,6.084,149.424
C09755=1139.932,-79.630,-45.398,178.881,6.083,149.425
C09756=1139.937,-79.880,-45.387,178.879,6.083,149.425
C09757=1139.942,-80.130,-45.377,178.877,6.082,149.426
C09758=1139.948,-80.380,-45.368,178.874,6.082,149.427
C09759=1139.953,-80.629,-45.358,178.873,6.082,149.427
C09760=1139.958,-80.879,-45.348,178.870,6.081,149.427
C09761=1139.964,-81.129,-45.339,178.868,6.080,149.428
C09762=1139.968,-81.379,-45.329,178.866,6.079,149.428
C09763=1139.974,-81.628,-45.318,178.864,6.080,149.429
C09764=1139.980,-81.878,-45.309,178.862,6.079,149.430
C09765=1139.985,-82.128,-45.299,178.860,6.078,149.430
C09766=1139.991,-82.378,-45.290,178.857,6.078,149.431
C09767=1139.995,-82.627,-45.280,178.856,6.078,149.431
C09768=1140.000,-82.877,-45.270,178.853,6.077,149.432
C09769=1140.006,-83.127,-45.260,178.851,6.076,149.432
C09770=1140.011,-83.377,-45.250,178.849,6.076,149.433
C09771=1140.017,-83.627,-45.241,178.847,6.076,149.433
C09772=1140.022,-83.876,-45.231,178.845,6.075,149.434
C09773=1140.028,-84.126,-45.221,178.842,6.075,149.434
C09774=1140.033,-84.375,-45.212,178.841,6.075,149.435
C09775=1140.038,-84.625,-45.202,178.839,6.074,149.435
C09776=1140.044,-84.876,-45.192,178.836,6.073,149.436
C09777=1140.048,-85.125,-45.183,178.835,6.073,149.436
C09778=1140.054,-85.375,-45.173,178.832,6.073,149.437
C09779=1140.059,-85.624,-45.163,178.830,6.072,149.438
C09780=1140.065,-85.874,-45.153,178.828,6.071,149.438
C09781=1140.070,-86.124,-45.144,178.826,6.071,149.439
C09782=1140.076,-86.373,-45.134,178.824,6.071,149.439
C09783=1140.081,-86.623,-45.125,178.821,6.070,149.440
C09784=1140.086,-86.873,-45.115,178.820,6.070,149.440
C09785=1140.091,-87.123,-45.106,178.817,6.069,149.441
C09786=1140.097,-87.373,-45.096,178.815,6.069,149.441
C09787=1140.102,-87.623,-45.087,178.814,6.069,149.442
C09788=1140.107,-87.872,-45.076,178.811,6.068,149.442
C09789=1140.112,-88.122,-45.068,178.809,6.068,149.443
C09790=1140.118,-88.372,-45.057,178.807,6.067,149.443
C09791=1140.123,-88.622,-45.048,178.805,6.067,149.444
C09792=1140.128,-88.871,-45.040,178.803,6.066,149.444
C09793=1140.134,-89.121,-45.029,178.801,6.065,149.445
C09794=1140.139,-89.371,-45.020,178.799,6.066,149.446
C09795=1140.145,-89.620,-45.010,178.796,6.065,149.446
C09796=1140.150,-89.870,-45.001,178.794,6.064,149.446
C09797=1140.156,-90.120,-44.991,178.793,6.064,149.447
C09798=1140.161,-90.370,-44.982,178.790,6.064,149.447
C09799=1140.167,-90.620,-44.973,178.788,6.063,149.448
C09800=1140.171,-90.869,-44.963,178.786,6.063,149.449
C09801=1140.177,-91.119,-44.954,178.784,6.062,149.449
C09802=1140.182,-91.369,-44.944,178.782,6.062,149.450
C09803=1140.187,-91.619,-44.935,178.780,6.062,149.450
C09804=1140.193,-91.869,-44.925,178.778,6.061,149.451
C09805=1140.198,-92.118,-44.916,178.775,6.061,149.451
C09806=1140.203,-92.368,-44.907,178.774,6.061,149.452
C09807=1140.209,-92.618,-44.897,178.771,6.060,149.452
C09808=1140.213,-92.868,-44.888,178.769,6.059,149.453
C09809=1140.219,-93.118,-44.878,178.768,6.059,149.453
C09810=1140.225,-93.368,-44.869,178.765,6.058,149.454
C09811=1140.229,-93.617,-44.860,178.763,6.058,149.454
C09812=1140.235,-93.867,-44.850,178.761,6.058,149.455
C09813=1140.240,-94.117,-44.841,178.759,6.057,149.455
C09814=1140.246,-94.366,-44.831,178.757,6.057,149.456
C09815=1140.251,-94.616,-44.822,178.755,6.057,149.456
C09816=1140.256,-94.866,-44.813,178.753,6.056,149.457
C09817=1140.262,-95.116,-44.803,178.751,6.055,149.457
C09818=1140.267,-95.365,-44.794,178.749,6.056,149.458
C09819=1140.272,-95.615,-44.785,178.747,6.055,149.459
C09820=1140.279,-95.865,-44.776,178.744,6.054,149.459
C09821=1140.284,-96.114,-44.767,178.743,6.054,149.460
C09822=1140.289,-96.364,-44.758,178.741,6.053,149.460
C09823=1140.295,-96.614,-44.748,178.738,6.053,149.460
C09824=1140.300,-96.864,-44.739,178.736,6.053,149.461
C09825=1140.305,-97.113,-44.730,178.734,6.052,149.462
C09826=1140.311,-97.363,-44.720,178.732,6.051,149.462
C09827=1140.316,-97.613,-44.711,178.730,6.051,149.463
C09828=1140.321,-97.863,-44.702,178.728,6.051,149.463
C09829=1140.326,-98.113,-44.693,178.726,6.050,149.464
C09830=1140.332,-98.362,-44.683,178.724,6.050,149.464
C09831=1140.337,-98.612,-44.674,178.722,6.050,149.465
C09832=1140.342,-98.862,-44.665,178.720,6.050,149.465
C09833=1140.348,-99.112,-44.656,178.718,6.049,149.466
C09834=1140.353,-99.362,-44.647,178.716,6.048,149.466
C09835=1140.358,-99.611,-44.637,178.714,6.048,149.467
C09836=1140.364,-99.860,-44.629,178.712,6.047,149.467
C09837=1140.370,-100.111,-44.619,178.710,6.047,149.468
C09838=1140.375,-100.360,-44.611,178.708,6.047,149.468
C09839=1140.380,-100.610,-44.602,178.705,6.046,149.469
C09840=1140.385,-100.860,-44.593,178.703,6.046,149.469
C09841=1140.391,-101.110,-44.583,178.702,6.046,149.470
C09842=1140.396,-101.360,-44.574,178.699,6.045,149.470
C09843=1140.401,-101.609,-44.565,178.698,6.045,149.471
C09844=1140.406,-101.859,-44.556,178.696,6.044,149.471
C09845=1140.412,-102.109,-44.547,178.693,6.043,149.472
C09846=1140.417,-102.359,-44.537,178.692,6.043,149.472
C09847=1140.424,-102.631,-44.528,178.689,6.043,149.473
C09848=1140.429,-102.903,-44.518,178.687,6.042,149.474
C09849=1140.435,-103.176,-44.509,178.685,6.042,149.474
C09850=1140.441,-103.448,-44.498,178.683,6.042,149.475
C09851=1140.446,-103.697,-44.489,178.680,6.041,149.475
C09852=1140.451,-103.947,-44.481,178.678,6.041,149.476
C09853=1140.457,-104.197,-44.471,178.677,6.041,149.476
C09854=1140.463,-104.447,-44.462,178.674,6.040,149.477
C09855=1140.468,-104.696,-44.454,178.673,6.040,149.477
C09856=1140.473,-104.946,-44.445,178.671,6.039,149.478
C09857=1140.478,-105.196,-44.436,178.668,6.039,149.478
C09858=1140.483,-105.446,-44.427,178.666,6.039,149.479
C09859=1140.488,-105.696,-44.418,178.664,6.038,149.479
C09860=1140.495,-105.945,-44.409,178.662,6.037,149.480
C09861=1140.500,-106.195,-44.400,178.660,6.037,149.480
C09862=1140.505,-106.445,-44.391,178.658,6.037,149.481
C09863=1140.510,-106.695,-44.382,178.657,6.037,149.481
C09864=1140.516,-106.945,-44.373,178.654,6.036,149.482
C09865=1140.521,-107.195,-44.364,178.652,6.035,149.482
C09866=1140.527,-107.444,-44.356,178.651,6.035,149.483
C09867=1140.532,-107.694,-44.347,178.648,6.035,149.483
C09868=1140.537,-107.943,-44.338,178.646,6.035,149.484
C09869=1140.543,-108.194,-44.329,178.644,6.034,149.484
C09870=1140.548,-108.443,-44.320,178.643,6.034,149.485
C09871=1140.553,-108.693,-44.311,178.640,6.033,149.485
C09872=1140.559,-108.943,-44.303,178.638,6.033,149.486
C09873=1140.564,-109.193,-44.294,178.637,6.033,149.486
C09874=1140.570,-109.443,-44.285,178.634,6.032,149.487
C09875=1140.575,-109.693,-44.276,178.633,6.032,149.487
C09876=1140.580,-109.942,-44.267,178.631,6.031,149.488
C09877=1140.586,-110.192,-44.259,178.628,6.031,149.488
C09878=1140.591,-110.441,-44.250,178.627,6.031,149.489
C09879=1140.596,-110.691,-44.241,178.624,6.030,149.490
C09880=1140.601,-110.941,-44.232,178.623,6.030,149.490
C09881=1140.607,-111.191,-44.224,178.620,6.030,149.490
C09882=1140.612,-111.441,-44.215,178.618,6.029,149.491
C09883=1140.618,-111.691,-44.207,178.617,6.029,149.491
C09884=1140.623,-111.940,-44.198,178.614,6.028,149.492
C09885=1140.628,-112.190,-44.189,178.613,6.028,149.492
C09886=1140.634,-112.440,-44.180,178.611,6.027,149.493
C09887=1140.640,-112.690,-44.171,178.609,6.027,149.493
C09888=1140.645,-112.940,-44.163,178.607,6.027,149.494
C09889=1140.651,-113.189,-44.154,178.605,6.026,149.494
C09890=1140.656,-113.439,-44.145,178.603,6.026,149.495
C09891=1140.661,-113.689,-44.136,178.601,6.025,149.495
C09892=1140.666,-113.939,-44.127,178.599,6.025,149.496
C09893=1140.672,-114.189,-44.119,178.596,6.025,149.497
C09894=1140.678,-114.438,-44.111,178.595,6.025,149.497
C09895=1140.683,-114.688,-44.102,178.593,6.024,149.498
C09896=1140.687,-114.938,-44.093,178.590,6.023,149.498
C09897=1140.693,-115.188,-44.086,178.589,6.023,149.499
C09898=1140.698,-115.437,-44.077,178.587,6.023,149.499
C09899=1140.704,-115.687,-44.068,178.585,6.023,149.499
C09900=1140.709,-115.936,-44.059,178.583,6.022,149.500
C09901=1140.715,-116.187,-44.051,178.581,6.022,149.500
C09902=1140.720,-116.437,-44.042,178.579,6.021,149.501
C09903=1140.725,-116.687,-44.033,178.578,6.021,149.501
C09904=1140.731,-116.936,-44.025,178.575,6.021,149.502
C09905=1140.736,-117.186,-44.017,178.573,6.020,149.502
C09906=1140.741,-117.436,-44.008,178.572,6.020,149.503
C09907=1140.747,-117.685,-43.999,178.569,6.019,149.503
C09908=1140.753,-117.936,-43.991,178.568,6.019,149.504
C09909=1140.758,-118.186,-43.982,178.566,6.018,149.504
C09910=1140.764,-118.435,-43.973,178.564,6.018,149.505
C09911=1140.769,-118.685,-43.965,178.562,6.018,149.505
C09912=1140.774,-118.935,-43.956,178.560,6.018,149.506
C09913=1140.779,-119.184,-43.948,178.558,6.017,149.506
C09914=1140.785,-119.434,-43.940,178.556,6.017,149.507
C09915=1140.790,-119.684,-43.931,178.554,6.016,149.507
C09916=1140.796,-119.933,-43.923,178.551,6.016,149.508
C09917=1140.801,-120.184,-43.915,178.550,6.016,149.508
C09918=1140.806,-120.434,-43.906,178.548,6.015,149.509
C09919=1140.812,-120.683,-43.897,178.546,6.015,149.509
C09920=1140.818,-120.933,-43.889,178.544,6.015,149.510
C09921=1140.822,-121.183,-43.881,178.542,6.015,149.510
C09922=1140.828,-121.433,-43.873,178.540,6.014,149.511
C09923=1140.833,-121.682,-43.864,178.538,6.014,149.511
C09924=1140.838,-121.932,-43.855,178.536,6.013,149.512
C09925=1140.845,-122.182,-43.847,178.535,6.013,149.512
C09926=1140.850,-122.432,-43.838,178.532,6.012,149.513
C09927=1140.854,-122.682,-43.831,178.531,6.013,149.513
C09928=1140.860,-122.931,-43.822,178.529,6.012,149.514
C09929=1140.865,-123.181,-43.813,178.527,6.012,149.514
C09930=1140.871,-123.431,-43.806,178.525,6.011,149.515
C09931=1140.877,-123.681,-43.797,178.523,6.010,149.515
C09932=1140.881,-123.931,-43.789,178.521,6.010,149.516
C09933=1140.887,-124.180,-43.781,178.519,6.010,149.516
C09934=1140.893,-124.430,-43.772,178.517,6.010,149.517
C09935=1140.898,-124.680,-43.764,178.515,6.009,149.517
C09936=1140.904,-124.930,-43.756,178.514,6.009,149.518
C09937=1140.908,-125.180,-43.747,178.511,6.008,149.518
C09938=1140.914,-125.429,-43.740,178.510,6.008,149.519
C09939=1140.919,-125.679,-43.731,178.508,6.008,149.519
C09940=1140.926,-125.929,-43.723,178.506,6.008,149.520
C09941=1140.931,-126.179,-43.714,178.504,6.007,149.520
C09942=1140.935,-126.429,-43.706,178.502,6.007,149.521
C09943=1140.941,-126.678,-43.698,178.500,6.006,149.521
C09944=1140.947,-126.929,-43.690,178.498,6.006,149.522
C09945=1140.952,-127.178,-43.681,178.496,6.005,149.522
C09946=1140.957,-127.428,-43.674,178.495,6.006,149.523
C09947=1140.962,-127.678,-43.665,178.492,6.005,149.523
C09948=1140.968,-127.928,-43.657,178.491,6.005,149.524
C09949=1140.974,-128.177,-43.648,178.489,6.004,149.524
C09950=1140.979,-128.427,-43.641,178.487,6.004,149.525
C09951=1140.559,-128.438,-43.684,178.484,6.007,149.526
C09952=1140.553,-128.189,-43.692,178.486,6.008,149.526
C09953=1140.547,-127.939,-43.701,178.487,6.008,149.525
C09954=1140.542,-127.689,-43.708,178.490,6.008,149.525
C09955=1140.537,-127.439,-43.716,178.491,6.008,149.524
C09956=1140.531,-127.190,-43.725,178.493,6.009,149.524
C09957=1140.525,-126.939,-43.733,178.495,6.009,149.523
C09958=1140.521,-126.690,-43.741,178.497,6.010,149.523
C09959=1140.515,-126.440,-43.749,178.499,6.010,149.522
C09960=1140.510,-126.190,-43.758,178.501,6.011,149.522
C09961=1140.504,-125.940,-43.766,178.502,6.011,149.522
C09962=1140.499,-125.691,-43.774,178.504,6.012,149.521
C09963=1140.493,-125.441,-43.782,178.506,6.012,149.521
C09964=1140.488,-125.191,-43.791,178.508,6.012,149.520
C09965=1140.482,-124.941,-43.799,178.510,6.012,149.520
C09966=1140.477,-124.691,-43.808,178.512,6.013,149.519
C09967=1140.472,-124.441,-43.815,178.513,6.013,149.519
C09968=1140.466,-124.192,-43.824,178.516,6.014,149.518
C09969=1140.461,-123.942,-43.832,178.517,6.014,149.518
C09970=1140.456,-123.692,-43.841,178.519,6.014,149.517
C09971=1140.449,-123.442,-43.849,178.521,6.014,149.517
C09972=1140.445,-123.192,-43.857,178.523,6.015,149.516
C09973=1140.440,-122.943,-43.866,178.525,6.016,149.516
C09974=1140.434,-122.693,-43.874,178.527,6.016,149.515
C09975=1140.429,-122.443,-43.883,178.529,6.017,149.515
C09976=1140.423,-122.193,-43.890,178.531,6.017,149.514
C09977=1140.417,-121.943,-43.899,178.534,6.017,149.513
C09978=1140.413,-121.693,-43.907,178.535,6.017,149.513
C09979=1140.407,-121.444,-43.915,178.537,6.018,149.513
C09980=1140.402,-121.194,-43.924,178.539,6.018,149.512
C09981=1140.396,-120.944,-43.932,178.541,6.018,149.512
C09982=1140.390,-120.695,-43.941,178.543,6.018,149.511
C09983=1140.385,-120.445,-43.950,178.545,6.019,149.511
C09984=1140.381,-120.195,-43.958,178.546,6.019,149.510
C09985=1140.375,-119.945,-43.966,178.549,6.020,149.510
C09986=1140.369,-119.695,-43.974,178.550,6.020,149.509
C09987=1140.364,-119.445,-43.983,178.552,6.020,149.509
C09988=1140.358,-119.196,-43.992,178.555,6.021,149.508
C09989=1140.353,-118.945,-44.000,178.556,6.021,149.508
C09990=1140.348,-118.696,-44.009,178.558,6.022,149.507
C09991=1140.342,-118.446,-44.017,178.560,6.022,149.507
C09992=1140.337,-118.196,-44.025,178.562,6.022,149.506
C09993=1140.331,-117.946,-44.034,178.564,6.022,149.506
C09994=1140.326,-117.697,-44.042,178.566,6.023,149.505
C09995=1140.321,-117.447,-44.050,178.568,6.023,149.505
C09996=1140.316,-117.197,-44.059,178.570,6.024,149.504
//INST
///DATE 2021/06/25 14:32
///ATTR SC,RW,RJ
////FRAME ROBOT
///GROUP1 RB1
NOP
MOVL C00000 V=800.0 PL=0
MOVL C00001 V=800.0 PL=0
MOVL C00002 V=800.0 PL=0
MOVL C00003 V=800.0 PL=0
MOVL C00004 V=800.0 PL=0
MOVL C00005 V=800.0 PL=0
MOVL C00006 V=800.0 PL=0
MOVL C00007 V=800.0 PL=0
MOVL C00008 V=800.0 PL=0
MOVL C00009 V=800.0 PL=0
MOVL C00010 V=800.0 PL=0
MOVL C00011 V=800.0 PL=0
MOVL C00012 V=800.0 PL=0
MOVL C00013 V=800.0 PL=0
MOVL C00014 V=800.0 PL=0
MOVL C00015 V=800.0 PL=0
MOVL C00016 V=800.0 PL=0
MOVL C00017 V=800.0 PL=0
MOVL C00018 V=800.0 PL=0
MOVL C00019 V=800.0 PL=0
MOVL C00020 V=800.0 PL=0
MOVL C00021 V=800.0 PL=0
MOVL C00022 V=800.0 PL=0
MOVL C00023 V=800.0 PL=0
MOVL C00024 V=800.0 PL=0
MOVL C00025 V=800.0 PL=0
MOVL C00026 V=800.0 PL=0
MOVL C00027 V=800.0 PL=0
MOVL C00028 V=800.0 PL=0
MOVL C00029 V=800.0 PL=0
MOVL C00030 V=800.0 PL=0
MOVL C00031 V=800.0 PL=0
MOVL C00032 V=800.0 PL=0
MOVL C00033 V=800.0 PL=0
MOVL C00034 V=800.0 PL=0
MOVL C00035 V=800.0 PL=0
MOVL C00036 V=800.0 PL=0
MOVL C00037 V=800.0 PL=0
MOVL C00038 V=800.0 PL=0
MOVL C00039 V=800.0 PL=0
MOVL C00040 V=800.0 PL=0
MOVL C00041 V=800.0 PL=0
MOVL C00042 V=800.0 PL=0
MOVL C00043 V=800.0 PL=0
MOVL C00044 V=800.0 PL=0
MOVL C00045 V=800.0 PL=0
MOVL C00046 V=800.0 PL=0
MOVL C00047 V=800.0 PL=0
MOVL C00048 V=800.0 PL=0
MOVL C00049 V=800.0 PL=0
MOVL C00050 V=800.0 PL=0
MOVL C00051 V=800.0 PL=0
MOVL C00052 V=800.0 PL=0
MOVL C00053 V=800.0 PL=0
MOVL C00054 V=800.0 PL=0
MOVL C00055 V=800.0 PL=0
MOVL C00056 V=800.0 PL=0
MOVL C00057 V=800.0 PL=0
MOVL C00058 V=800.0 PL=0
MOVL C00059 V=800.0 PL=0
MOVL C00060 V=800.0 PL=0
MOVL C00061 V=800.0 PL=0
MOVL C00062 V=800.0 PL=0
MOVL C00063 V=800.0 PL=0
MOVL C00064 V=800.0 PL=0
MOVL C00065 V=800.0 PL=0
MOVL C00066 V=800.0 PL=0
MOVL C00067 V=800.0 PL=0
MOVL C00068 V=800.0 PL=0
MOVL C00069 V=800.0 PL=0
MOVL C00070 V=800.0 PL=0
MOVL C00071 V=800.0 PL=0
MOVL C00072 V=800.0 PL=0
MOVL C00073 V=800.0 PL=0
MOVL C00074 V=800.0 PL=0
MOVL C00075 V=800.0 PL=0
MOVL C00076 V=800.0 PL=0
MOVL C00077 V=800.0 PL=0
MOVL C00078 V=800.0 PL=0
MOVL C00079 V=800.0 PL=0
MOVL C00080 V=800.0 PL=0
MOVL C00081 V=800.0 PL=0
MOVL C00082 V=800.0 PL=0
MOVL C00083 V=800.0 PL=0
MOVL C00084 V=800.0 PL=0
MOVL C00085 V=800.0 PL=0
MOVL C00086 V=800.0 PL=0
MOVL C00087 V=800.0 PL=0
MOVL C00088 V=800.0 PL=0
MOVL C00089 V=800.0 PL=0
MOVL C00090 V=800.0 PL=0
MOVL C00091 V=800.0 PL=0
MOVL C00092 V=800.0 PL=0
MOVL C00093 V=800.0 PL=0
MOVL C00094 V=800.0 PL=0
MOVL C00095 V=800.0 PL=0
MOVL C00096 V=800.0 PL=0
MOVL C00097 V=800.0 PL=0
MOVL C00098 V=800.0 PL=0
MOVL C00099 V=800.0 PL=0
MOVL C00100 V=800.0 PL=0
MOVL C00101 V=800.0 PL=0
MOVL C00102 V=800.0 PL=0
MOVL C00103 V=800.0 PL=0
MOVL C00104 V=800.0 PL=0
MOVL C00105 V=800.0 PL=0
MOVL C00106 V=800.0 PL=0
MOVL C00107 V=800.0 PL=0
MOVL C00108 V=800.0 PL=0
MOVL C00109 V=800.0 PL=0
MOVL C00110 V=800.0 PL=0
MOVL C00111 V=800.0 PL=0
MOVL C00112 V=800.0 PL=0
MOVL C00113 V=800.0 PL=0
MOVL C00114 V=800.0 PL=0
MOVL C00115 V=800.0 PL=0
MOVL C00116 V=800.0 PL=0
MOVL C00117 V=800.0 PL=0
MOVL C00118 V=800.0 PL=0
MOVL C00119 V=800.0 PL=0
MOVL C00120 V=800.0 PL=0
MOVL C00121 V=800.0 PL=0
MOVL C00122 V=800.0 PL=0
MOVL C00123 V=800.0 PL=0
MOVL C00124 V=800.0 PL=0
MOVL C00125 V=800.0 PL=0
MOVL C00126 V=800.0 PL=0
MOVL C00127 V=800.0 PL=0
MOVL C00128 V=800.0 PL=0
MOVL C00129 V=800.0 PL=0
MOVL C00130 V=800.0 PL=0
MOVL C00131 V=800.0 PL=0
MOVL C00132 V=800.0 PL=0
MOVL C00133 V=800.0 PL=0
MOVL C00134 V=800.0 PL=0
MOVL C00135 V=800.0 PL=0
MOVL C00136 V=800.0 PL=0
MOVL C00137 V=800.0 PL=0
MOVL C00138 V=800.0 PL=0
MOVL C00139 V=800.0 PL=0
MOVL C00140 V=800.0 PL=0
MOVL C00141 V=800.0 PL=0
MOVL C00142 V=800.0 PL=0
MOVL C00143 V=800.0 PL=0
MOVL C00144 V=800.0 PL=0
MOVL C00145 V=800.0 PL=0
MOVL C00146 V=800.0 PL=0
MOVL C00147 V=800.0 PL=0
MOVL C00148 V=800.0 PL=0
MOVL C00149 V=800.0 PL=0
MOVL C00150 V=800.0 PL=0
MOVL C00151 V=800.0 PL=0
MOVL C00152 V=800.0 PL=0
MOVL C00153 V=800.0 PL=0
MOVL C00154 V=800.0 PL=0
MOVL C00155 V=800.0 PL=0
MOVL C00156 V=800.0 PL=0
MOVL C00157 V=800.0 PL=0
MOVL C00158 V=800.0 PL=0
MOVL C00159 V=800.0 PL=0
MOVL C00160 V=800.0 PL=0
MOVL C00161 V=800.0 PL=0
MOVL C00162 V=800.0 PL=0
MOVL C00163 V=800.0 PL=0
MOVL C00164 V=800.0 PL=0
MOVL C00165 V=800.0 PL=0
MOVL C00166 V=800.0 PL=0
MOVL C00167 V=800.0 PL=0
MOVL C00168 V=800.0 PL=0
MOVL C00169 V=800.0 PL=0
MOVL C00170 V=800.0 PL=0
MOVL C00171 V=800.0 PL=0
MOVL C00172 V=800.0 PL=0
MOVL C00173 V=800.0 PL=0
MOVL C00174 V=800.0 PL=0
MOVL C00175 V=800.0 PL=0
MOVL C00176 V=800.0 PL=0
MOVL C00177 V=800.0 PL=0
MOVL C00178 V=800.0 PL=0
MOVL C00179 V=800.0 PL=0
MOVL C00180 V=800.0 PL=0
MOVL C00181 V=800.0 PL=0
MOVL C00182 V=800.0 PL=0
MOVL C00183 V=800.0 PL=0
MOVL C00184 V=800.0 PL=0
MOVL C00185 V=800.0 PL=0
MOVL C00186 V=800.0 PL=0
MOVL C00187 V=800.0 PL=0
MOVL C00188 V=800.0 PL=0
MOVL C00189 V=800.0 PL=0
MOVL C00190 V=800.0 PL=0
MOVL C00191 V=800.0 PL=0
MOVL C00192 V=800.0 PL=0
MOVL C00193 V=800.0 PL=0
MOVL C00194 V=800.0 PL=0
MOVL C00195 V=800.0 PL=0
MOVL C00196 V=800.0 PL=0
MOVL C00197 V=800.0 PL=0
MOVL C00198 V=800.0 PL=0
MOVL C00199 V=800.0 PL=0
MOVL C00200 V=800.0 PL=0
MOVL C00201 V=800.0 PL=0
MOVL C00202 V=800.0 PL=0
MOVL C00203 V=800.0 PL=0
MOVL C00204 V=800.0 PL=0
MOVL C00205 V=800.0 PL=0
MOVL C00206 V=800.0 PL=0
MOVL C00207 V=800.0 PL=0
MOVL C00208 V=800.0 PL=0
MOVL C00209 V=800.0 PL=0
MOVL C00210 V=800.0 PL=0
MOVL C00211 V=800.0 PL=0
MOVL C00212 V=800.0 PL=0
MOVL C00213 V=800.0 PL=0
MOVL C00214 V=800.0 PL=0
MOVL C00215 V=800.0 PL=0
MOVL C00216 V=800.0 PL=0
MOVL C00217 V=800.0 PL=0
MOVL C00218 V=800.0 PL=0
MOVL C00219 V=800.0 PL=0
MOVL C00220 V=800.0 PL=0
MOVL C00221 V=800.0 PL=0
MOVL C00222 V=800.0 PL=0
MOVL C00223 V=800.0 PL=0
MOVL C00224 V=800.0 PL=0
MOVL C00225 V=800.0 PL=0
MOVL C00226 V=800.0 PL=0
MOVL C00227 V=800.0 PL=0
MOVL C00228 V=800.0 PL=0
MOVL C00229 V=800.0 PL=0
MOVL C00230 V=800.0 PL=0
MOVL C00231 V=800.0 PL=0
MOVL C00232 V=800.0 PL=0
MOVL C00233 V=800.0 PL=0
MOVL C00234 V=800.0 PL=0
MOVL C00235 V=800.0 PL=0
MOVL C00236 V=800.0 PL=0
MOVL C00237 V=800.0 PL=0
MOVL C00238 V=800.0 PL=0
MOVL C00239 V=800.0 PL=0
MOVL C00240 V=800.0 PL=0
MOVL C00241 V=800.0 PL=0
MOVL C00242 V=800.0 PL=0
MOVL C00243 V=800.0 PL=0
MOVL C00244 V=800.0 PL=0
MOVL C00245 V=800.0 PL=0
MOVL C00246 V=800.0 PL=0
MOVL C00247 V=800.0 PL=0
MOVL C00248 V=800.0 PL=0
MOVL C00249 V=800.0 PL=0
MOVL C00250 V=800.0 PL=0
MOVL C00251 V=800.0 PL=0
MOVL C00252 V=800.0 PL=0
MOVL C00253 V=800.0 PL=0
MOVL C00254 V=800.0 PL=0
MOVL C00255 V=800.0 PL=0
MOVL C00256 V=800.0 PL=0
MOVL C00257 V=800.0 PL=0
MOVL C00258 V=800.0 PL=0
MOVL C00259 V=800.0 PL=0
MOVL C00260 V=800.0 PL=0
MOVL C00261 V=800.0 PL=0
MOVL C00262 V=800.0 PL=0
MOVL C00263 V=800.0 PL=0
MOVL C00264 V=800.0 PL=0
MOVL C00265 V=800.0 PL=0
MOVL C00266 V=800.0 PL=0
MOVL C00267 V=800.0 PL=0
MOVL C00268 V=800.0 PL=0
MOVL C00269 V=800.0 PL=0
MOVL C00270 V=800.0 PL=0
MOVL C00271 V=800.0 PL=0
MOVL C00272 V=800.0 PL=0
MOVL C00273 V=800.0 PL=0
MOVL C00274 V=800.0 PL=0
MOVL C00275 V=800.0 PL=0
MOVL C00276 V=800.0 PL=0
MOVL C00277 V=800.0 PL=0
MOVL C00278 V=800.0 PL=0
MOVL C00279 V=800.0 PL=0
MOVL C00280 V=800.0 PL=0
MOVL C00281 V=800.0 PL=0
MOVL C00282 V=800.0 PL=0
MOVL C00283 V=800.0 PL=0
MOVL C00284 V=800.0 PL=0
MOVL C00285 V=800.0 PL=0
MOVL C00286 V=800.0 PL=0
MOVL C00287 V=800.0 PL=0
MOVL C00288 V=800.0 PL=0
MOVL C00289 V=800.0 PL=0
MOVL C00290 V=800.0 PL=0
MOVL C00291 V=800.0 PL=0
MOVL C00292 V=800.0 PL=0
MOVL C00293 V=800.0 PL=0
MOVL C00294 V=800.0 PL=0
MOVL C00295 V=800.0 PL=0
MOVL C00296 V=800.0 PL=0
MOVL C00297 V=800.0 PL=0
MOVL C00298 V=800.0 PL=0
MOVL C00299 V=800.0 PL=0
MOVL C00300 V=800.0 PL=0
MOVL C00301 V=800.0 PL=0
MOVL C00302 V=800.0 PL=0
MOVL C00303 V=800.0 PL=0
MOVL C00304 V=800.0 PL=0
MOVL C00305 V=800.0 PL=0
MOVL C00306 V=800.0 PL=0
MOVL C00307 V=800.0 PL=0
MOVL C00308 V=800.0 PL=0
MOVL C00309 V=800.0 PL=0
MOVL C00310 V=800.0 PL=0
MOVL C00311 V=800.0 PL=0
MOVL C00312 V=800.0 PL=0
MOVL C00313 V=800.0 PL=0
MOVL C00314 V=800.0 PL=0
MOVL C00315 V=800.0 PL=0
MOVL C00316 V=800.0 PL=0
MOVL C00317 V=800.0 PL=0
MOVL C00318 V=800.0 PL=0
MOVL C00319 V=800.0 PL=0
MOVL C00320 V=800.0 PL=0
MOVL C00321 V=800.0 PL=0
MOVL C00322 V=800.0 PL=0
MOVL C00323 V=800.0 PL=0
MOVL C00324 V=800.0 PL=0
MOVL C00325 V=800.0 PL=0
MOVL C00326 V=800.0 PL=0
MOVL C00327 V=800.0 PL=0
MOVL C00328 V=800.0 PL=0
MOVL C00329 V=800.0 PL=0
MOVL C00330 V=800.0 PL=0
MOVL C00331 V=800.0 PL=0
MOVL C00332 V=800.0 PL=0
MOVL C00333 V=800.0 PL=0
MOVL C00334 V=800.0 PL=0
MOVL C00335 V=800.0 PL=0
MOVL C00336 V=800.0 PL=0
MOVL C00337 V=800.0 PL=0
MOVL C00338 V=800.0 PL=0
MOVL C00339 V=800.0 PL=0
MOVL C00340 V=800.0 PL=0
MOVL C00341 V=800.0 PL=0
MOVL C00342 V=800.0 PL=0
MOVL C00343 V=800.0 PL=0
MOVL C00344 V=800.0 PL=0
MOVL C00345 V=800.0 PL=0
MOVL C00346 V=800.0 PL=0
MOVL C00347 V=800.0 PL=0
MOVL C00348 V=800.0 PL=0
MOVL C00349 V=800.0 PL=0
MOVL C00350 V=800.0 PL=0
MOVL C00351 V=800.0 PL=0
MOVL C00352 V=800.0 PL=0
MOVL C00353 V=800.0 PL=0
MOVL C00354 V=800.0 PL=0
MOVL C00355 V=800.0 PL=0
MOVL C00356 V=800.0 PL=0
MOVL C00357 V=800.0 PL=0
MOVL C00358 V=800.0 PL=0
MOVL C00359 V=800.0 PL=0
MOVL C00360 V=800.0 PL=0
MOVL C00361 V=800.0 PL=0
MOVL C00362 V=800.0 PL=0
MOVL C00363 V=800.0 PL=0
MOVL C00364 V=800.0 PL=0
MOVL C00365 V=800.0 PL=0
MOVL C00366 V=800.0 PL=0
MOVL C00367 V=800.0 PL=0
MOVL C00368 V=800.0 PL=0
MOVL C00369 V=800.0 PL=0
MOVL C00370 V=800.0 PL=0
MOVL C00371 V=800.0 PL=0
MOVL C00372 V=800.0 PL=0
MOVL C00373 V=800.0 PL=0
MOVL C00374 V=800.0 PL=0
MOVL C00375 V=800.0 PL=0
MOVL C00376 V=800.0 PL=0
MOVL C00377 V=800.0 PL=0
MOVL C00378 V=800.0 PL=0
MOVL C00379 V=800.0 PL=0
MOVL C00380 V=800.0 PL=0
MOVL C00381 V=800.0 PL=0
MOVL C00382 V=800.0 PL=0
MOVL C00383 V=800.0 PL=0
MOVL C00384 V=800.0 PL=0
MOVL C00385 V=800.0 PL=0
MOVL C00386 V=800.0 PL=0
MOVL C00387 V=800.0 PL=0
MOVL C00388 V=800.0 PL=0
MOVL C00389 V=800.0 PL=0
MOVL C00390 V=800.0 PL=0
MOVL C00391 V=800.0 PL=0
MOVL C00392 V=800.0 PL=0
MOVL C00393 V=800.0 PL=0
MOVL C00394 V=800.0 PL=0
MOVL C00395 V=800.0 PL=0
MOVL C00396 V=800.0 PL=0
MOVL C00397 V=800.0 PL=0
MOVL C00398 V=800.0 PL=0
MOVL C00399 V=800.0 PL=0
MOVL C00400 V=800.0 PL=0
MOVL C00401 V=800.0 PL=0
MOVL C00402 V=800.0 PL=0
MOVL C00403 V=800.0 PL=0
MOVL C00404 V=800.0 PL=0
MOVL C00405 V=800.0 PL=0
MOVL C00406 V=800.0 PL=0
MOVL C00407 V=800.0 PL=0
MOVL C00408 V=800.0 PL=0
MOVL C00409 V=800.0 PL=0
MOVL C00410 V=800.0 PL=0
MOVL C00411 V=800.0 PL=0
MOVL C00412 V=800.0 PL=0
MOVL C00413 V=800.0 PL=0
MOVL C00414 V=800.0 PL=0
MOVL C00415 V=800.0 PL=0
MOVL C00416 V=800.0 PL=0
MOVL C00417 V=800.0 PL=0
MOVL C00418 V=800.0 PL=0
MOVL C00419 V=800.0 PL=0
MOVL C00420 V=800.0 PL=0
MOVL C00421 V=800.0 PL=0
MOVL C00422 V=800.0 PL=0
MOVL C00423 V=800.0 PL=0
MOVL C00424 V=800.0 PL=0
MOVL C00425 V=800.0 PL=0
MOVL C00426 V=800.0 PL=0
MOVL C00427 V=800.0 PL=0
MOVL C00428 V=800.0 PL=0
MOVL C00429 V=800.0 PL=0
MOVL C00430 V=800.0 PL=0
MOVL C00431 V=800.0 PL=0
MOVL C00432 V=800.0 PL=0
MOVL C00433 V=800.0 PL=0
MOVL C00434 V=800.0 PL=0
MOVL C00435 V=800.0 PL=0
MOVL C00436 V=800.0 PL=0
MOVL C00437 V=800.0 PL=0
MOVL C00438 V=800.0 PL=0
MOVL C00439 V=800.0 PL=0
MOVL C00440 V=800.0 PL=0
MOVL C00441 V=800.0 PL=0
MOVL C00442 V=800.0 PL=0
MOVL C00443 V=800.0 PL=0
MOVL C00444 V=800.0 PL=0
MOVL C00445 V=800.0 PL=0
MOVL C00446 V=800.0 PL=0
MOVL C00447 V=800.0 PL=0
MOVL C00448 V=800.0 PL=0
MOVL C00449 V=800.0 PL=0
MOVL C00450 V=800.0 PL=0
MOVL C00451 V=800.0 PL=0
MOVL C00452 V=800.0 PL=0
MOVL C00453 V=800.0 PL=0
MOVL C00454 V=800.0 PL=0
MOVL C00455 V=800.0 PL=0
MOVL C00456 V=800.0 PL=0
MOVL C00457 V=800.0 PL=0
MOVL C00458 V=800.0 PL=0
MOVL C00459 V=800.0 PL=0
MOVL C00460 V=800.0 PL=0
MOVL C00461 V=800.0 PL=0
MOVL C00462 V=800.0 PL=0
MOVL C00463 V=800.0 PL=0
MOVL C00464 V=800.0 PL=0
MOVL C00465 V=800.0 PL=0
MOVL C00466 V=800.0 PL=0
MOVL C00467 V=800.0 PL=0
MOVL C00468 V=800.0 PL=0
MOVL C00469 V=800.0 PL=0
MOVL C00470 V=800.0 PL=0
MOVL C00471 V=800.0 PL=0
MOVL C00472 V=800.0 PL=0
MOVL C00473 V=800.0 PL=0
MOVL C00474 V=800.0 PL=0
MOVL C00475 V=800.0 PL=0
MOVL C00476 V=800.0 PL=0
MOVL C00477 V=800.0 PL=0
MOVL C00478 V=800.0 PL=0
MOVL C00479 V=800.0 PL=0
MOVL C00480 V=800.0 PL=0
MOVL C00481 V=800.0 PL=0
MOVL C00482 V=800.0 PL=0
MOVL C00483 V=800.0 PL=0
MOVL C00484 V=800.0 PL=0
MOVL C00485 V=800.0 PL=0
MOVL C00486 V=800.0 PL=0
MOVL C00487 V=800.0 PL=0
MOVL C00488 V=800.0 PL=0
MOVL C00489 V=800.0 PL=0
MOVL C00490 V=800.0 PL=0
MOVL C00491 V=800.0 PL=0
MOVL C00492 V=800.0 PL=0
MOVL C00493 V=800.0 PL=0
MOVL C00494 V=800.0 PL=0
MOVL C00495 V=800.0 PL=0
MOVL C00496 V=800.0 PL=0
MOVL C00497 V=800.0 PL=0
MOVL C00498 V=800.0 PL=0
MOVL C00499 V=800.0 PL=0
MOVL C00500 V=800.0 PL=0
MOVL C00501 V=800.0 PL=0
MOVL C00502 V=800.0 PL=0
MOVL C00503 V=800.0 PL=0
MOVL C00504 V=800.0 PL=0
MOVL C00505 V=800.0 PL=0
MOVL C00506 V=800.0 PL=0
MOVL C00507 V=800.0 PL=0
MOVL C00508 V=800.0 PL=0
MOVL C00509 V=800.0 PL=0
MOVL C00510 V=800.0 PL=0
MOVL C00511 V=800.0 PL=0
MOVL C00512 V=800.0 PL=0
MOVL C00513 V=800.0 PL=0
MOVL C00514 V=800.0 PL=0
MOVL C00515 V=800.0 PL=0
MOVL C00516 V=800.0 PL=0
MOVL C00517 V=800.0 PL=0
MOVL C00518 V=800.0 PL=0
MOVL C00519 V=800.0 PL=0
MOVL C00520 V=800.0 PL=0
MOVL C00521 V=800.0 PL=0
MOVL C00522 V=800.0 PL=0
MOVL C00523 V=800.0 PL=0
MOVL C00524 V=800.0 PL=0
MOVL C00525 V=800.0 PL=0
MOVL C00526 V=800.0 PL=0
MOVL C00527 V=800.0 PL=0
MOVL C00528 V=800.0 PL=0
MOVL C00529 V=800.0 PL=0
MOVL C00530 V=800.0 PL=0
MOVL C00531 V=800.0 PL=0
MOVL C00532 V=800.0 PL=0
MOVL C00533 V=800.0 PL=0
MOVL C00534 V=800.0 PL=0
MOVL C00535 V=800.0 PL=0
MOVL C00536 V=800.0 PL=0
MOVL C00537 V=800.0 PL=0
MOVL C00538 V=800.0 PL=0
MOVL C00539 V=800.0 PL=0
MOVL C00540 V=800.0 PL=0
MOVL C00541 V=800.0 PL=0
MOVL C00542 V=800.0 PL=0
MOVL C00543 V=800.0 PL=0
MOVL C00544 V=800.0 PL=0
MOVL C00545 V=800.0 PL=0
MOVL C00546 V=800.0 PL=0
MOVL C00547 V=800.0 PL=0
MOVL C00548 V=800.0 PL=0
MOVL C00549 V=800.0 PL=0
MOVL C00550 V=800.0 PL=0
MOVL C00551 V=800.0 PL=0
MOVL C00552 V=800.0 PL=0
MOVL C00553 V=800.0 PL=0
MOVL C00554 V=800.0 PL=0
MOVL C00555 V=800.0 PL=0
MOVL C00556 V=800.0 PL=0
MOVL C00557 V=800.0 PL=0
MOVL C00558 V=800.0 PL=0
MOVL C00559 V=800.0 PL=0
MOVL C00560 V=800.0 PL=0
MOVL C00561 V=800.0 PL=0
MOVL C00562 V=800.0 PL=0
MOVL C00563 V=800.0 PL=0
MOVL C00564 V=800.0 PL=0
MOVL C00565 V=800.0 PL=0
MOVL C00566 V=800.0 PL=0
MOVL C00567 V=800.0 PL=0
MOVL C00568 V=800.0 PL=0
MOVL C00569 V=800.0 PL=0
MOVL C00570 V=800.0 PL=0
MOVL C00571 V=800.0 PL=0
MOVL C00572 V=800.0 PL=0
MOVL C00573 V=800.0 PL=0
MOVL C00574 V=800.0 PL=0
MOVL C00575 V=800.0 PL=0
MOVL C00576 V=800.0 PL=0
MOVL C00577 V=800.0 PL=0
MOVL C00578 V=800.0 PL=0
MOVL C00579 V=800.0 PL=0
MOVL C00580 V=800.0 PL=0
MOVL C00581 V=800.0 PL=0
MOVL C00582 V=800.0 PL=0
MOVL C00583 V=800.0 PL=0
MOVL C00584 V=800.0 PL=0
MOVL C00585 V=800.0 PL=0
MOVL C00586 V=800.0 PL=0
MOVL C00587 V=800.0 PL=0
MOVL C00588 V=800.0 PL=0
MOVL C00589 V=800.0 PL=0
MOVL C00590 V=800.0 PL=0
MOVL C00591 V=800.0 PL=0
MOVL C00592 V=800.0 PL=0
MOVL C00593 V=800.0 PL=0
MOVL C00594 V=800.0 PL=0
MOVL C00595 V=800.0 PL=0
MOVL C00596 V=800.0 PL=0
MOVL C00597 V=800.0 PL=0
MOVL C00598 V=800.0 PL=0
MOVL C00599 V=800.0 PL=0
MOVL C00600 V=800.0 PL=0
MOVL C00601 V=800.0 PL=0
MOVL C00602 V=800.0 PL=0
MOVL C00603 V=800.0 PL=0
MOVL C00604 V=800.0 PL=0
MOVL C00605 V=800.0 PL=0
MOVL C00606 V=800.0 PL=0
MOVL C00607 V=800.0 PL=0
MOVL C00608 V=800.0 PL=0
MOVL C00609 V=800.0 PL=0
MOVL C00610 V=800.0 PL=0
MOVL C00611 V=800.0 PL=0
MOVL C00612 V=800.0 PL=0
MOVL C00613 V=800.0 PL=0
MOVL C00614 V=800.0 PL=0
MOVL C00615 V=800.0 PL=0
MOVL C00616 V=800.0 PL=0
MOVL C00617 V=800.0 PL=0
MOVL C00618 V=800.0 PL=0
MOVL C00619 V=800.0 PL=0
MOVL C00620 V=800.0 PL=0
MOVL C00621 V=800.0 PL=0
MOVL C00622 V=800.0 PL=0
MOVL C00623 V=800.0 PL=0
MOVL C00624 V=800.0 PL=0
MOVL C00625 V=800.0 PL=0
MOVL C00626 V=800.0 PL=0
MOVL C00627 V=800.0 PL=0
MOVL C00628 V=800.0 PL=0
MOVL C00629 V=800.0 PL=0
MOVL C00630 V=800.0 PL=0
MOVL C00631 V=800.0 PL=0
MOVL C00632 V=800.0 PL=0
MOVL C00633 V=800.0 PL=0
MOVL C00634 V=800.0 PL=0
MOVL C00635 V=800.0 PL=0
MOVL C00636 V=800.0 PL=0
MOVL C00637 V=800.0 PL=0
MOVL C00638 V=800.0 PL=0
MOVL C00639 V=800.0 PL=0
MOVL C00640 V=800.0 PL=0
MOVL C00641 V=800.0 PL=0
MOVL C00642 V=800.0 PL=0
MOVL C00643 V=800.0 PL=0
MOVL C00644 V=800.0 PL=0
MOVL C00645 V=800.0 PL=0
MOVL C00646 V=800.0 PL=0
MOVL C00647 V=800.0 PL=0
MOVL C00648 V=800.0 PL=0
MOVL C00649 V=800.0 PL=0
MOVL C00650 V=800.0 PL=0
MOVL C00651 V=800.0 PL=0
MOVL C00652 V=800.0 PL=0
MOVL C00653 V=800.0 PL=0
MOVL C00654 V=800.0 PL=0
MOVL C00655 V=800.0 PL=0
MOVL C00656 V=800.0 PL=0
MOVL C00657 V=800.0 PL=0
MOVL C00658 V=800.0 PL=0
MOVL C00659 V=800.0 PL=0
MOVL C00660 V=800.0 PL=0
MOVL C00661 V=800.0 PL=0
MOVL C00662 V=800.0 PL=0
MOVL C00663 V=800.0 PL=0
MOVL C00664 V=800.0 PL=0
MOVL C00665 V=800.0 PL=0
MOVL C00666 V=800.0 PL=0
MOVL C00667 V=800.0 PL=0
MOVL C00668 V=800.0 PL=0
MOVL C00669 V=800.0 PL=0
MOVL C00670 V=800.0 PL=0
MOVL C00671 V=800.0 PL=0
MOVL C00672 V=800.0 PL=0
MOVL C00673 V=800.0 PL=0
MOVL C00674 V=800.0 PL=0
MOVL C00675 V=800.0 PL=0
MOVL C00676 V=800.0 PL=0
MOVL C00677 V=800.0 PL=0
MOVL C00678 V=800.0 PL=0
MOVL C00679 V=800.0 PL=0
MOVL C00680 V=800.0 PL=0
MOVL C00681 V=800.0 PL=0
MOVL C00682 V=800.0 PL=0
MOVL C00683 V=800.0 PL=0
MOVL C00684 V=800.0 PL=0
MOVL C00685 V=800.0 PL=0
MOVL C00686 V=800.0 PL=0
MOVL C00687 V=800.0 PL=0
MOVL C00688 V=800.0 PL=0
MOVL C00689 V=800.0 PL=0
MOVL C00690 V=800.0 PL=0
MOVL C00691 V=800.0 PL=0
MOVL C00692 V=800.0 PL=0
MOVL C00693 V=800.0 PL=0
MOVL C00694 V=800.0 PL=0
MOVL C00695 V=800.0 PL=0
MOVL C00696 V=800.0 PL=0
MOVL C00697 V=800.0 PL=0
MOVL C00698 V=800.0 PL=0
MOVL C00699 V=800.0 PL=0
MOVL C00700 V=800.0 PL=0
MOVL C00701 V=800.0 PL=0
MOVL C00702 V=800.0 PL=0
MOVL C00703 V=800.0 PL=0
MOVL C00704 V=800.0 PL=0
MOVL C00705 V=800.0 PL=0
MOVL C00706 V=800.0 PL=0
MOVL C00707 V=800.0 PL=0
MOVL C00708 V=800.0 PL=0
MOVL C00709 V=800.0 PL=0
MOVL C00710 V=800.0 PL=0
MOVL C00711 V=800.0 PL=0
MOVL C00712 V=800.0 PL=0
MOVL C00713 V=800.0 PL=0
MOVL C00714 V=800.0 PL=0
MOVL C00715 V=800.0 PL=0
MOVL C00716 V=800.0 PL=0
MOVL C00717 V=800.0 PL=0
MOVL C00718 V=800.0 PL=0
MOVL C00719 V=800.0 PL=0
MOVL C00720 V=800.0 PL=0
MOVL C00721 V=800.0 PL=0
MOVL C00722 V=800.0 PL=0
MOVL C00723 V=800.0 PL=0
MOVL C00724 V=800.0 PL=0
MOVL C00725 V=800.0 PL=0
MOVL C00726 V=800.0 PL=0
MOVL C00727 V=800.0 PL=0
MOVL C00728 V=800.0 PL=0
MOVL C00729 V=800.0 PL=0
MOVL C00730 V=800.0 PL=0
MOVL C00731 V=800.0 PL=0
MOVL C00732 V=800.0 PL=0
MOVL C00733 V=800.0 PL=0
MOVL C00734 V=800.0 PL=0
MOVL C00735 V=800.0 PL=0
MOVL C00736 V=800.0 PL=0
MOVL C00737 V=800.0 PL=0
MOVL C00738 V=800.0 PL=0
MOVL C00739 V=800.0 PL=0
MOVL C00740 V=800.0 PL=0
MOVL C00741 V=800.0 PL=0
MOVL C00742 V=800.0 PL=0
MOVL C00743 V=800.0 PL=0
MOVL C00744 V=800.0 PL=0
MOVL C00745 V=800.0 PL=0
MOVL C00746 V=800.0 PL=0
MOVL C00747 V=800.0 PL=0
MOVL C00748 V=800.0 PL=0
MOVL C00749 V=800.0 PL=0
MOVL C00750 V=800.0 PL=0
MOVL C00751 V=800.0 PL=0
MOVL C00752 V=800.0 PL=0
MOVL C00753 V=800.0 PL=0
MOVL C00754 V=800.0 PL=0
MOVL C00755 V=800.0 PL=0
MOVL C00756 V=800.0 PL=0
MOVL C00757 V=800.0 PL=0
MOVL C00758 V=800.0 PL=0
MOVL C00759 V=800.0 PL=0
MOVL C00760 V=800.0 PL=0
MOVL C00761 V=800.0 PL=0
MOVL C00762 V=800.0 PL=0
MOVL C00763 V=800.0 PL=0
MOVL C00764 V=800.0 PL=0
MOVL C00765 V=800.0 PL=0
MOVL C00766 V=800.0 PL=0
MOVL C00767 V=800.0 PL=0
MOVL C00768 V=800.0 PL=0
MOVL C00769 V=800.0 PL=0
MOVL C00770 V=800.0 PL=0
MOVL C00771 V=800.0 PL=0
MOVL C00772 V=800.0 PL=0
MOVL C00773 V=800.0 PL=0
MOVL C00774 V=800.0 PL=0
MOVL C00775 V=800.0 PL=0
MOVL C00776 V=800.0 PL=0
MOVL C00777 V=800.0 PL=0
MOVL C00778 V=800.0 PL=0
MOVL C00779 V=800.0 PL=0
MOVL C00780 V=800.0 PL=0
MOVL C00781 V=800.0 PL=0
MOVL C00782 V=800.0 PL=0
MOVL C00783 V=800.0 PL=0
MOVL C00784 V=800.0 PL=0
MOVL C00785 V=800.0 PL=0
MOVL C00786 V=800.0 PL=0
MOVL C00787 V=800.0 PL=0
MOVL C00788 V=800.0 PL=0
MOVL C00789 V=800.0 PL=0
MOVL C00790 V=800.0 PL=0
MOVL C00791 V=800.0 PL=0
MOVL C00792 V=800.0 PL=0
MOVL C00793 V=800.0 PL=0
MOVL C00794 V=800.0 PL=0
MOVL C00795 V=800.0 PL=0
MOVL C00796 V=800.0 PL=0
MOVL C00797 V=800.0 PL=0
MOVL C00798 V=800.0 PL=0
MOVL C00799 V=800.0 PL=0
MOVL C00800 V=800.0 PL=0
MOVL C00801 V=800.0 PL=0
MOVL C00802 V=800.0 PL=0
MOVL C00803 V=800.0 PL=0
MOVL C00804 V=800.0 PL=0
MOVL C00805 V=800.0 PL=0
MOVL C00806 V=800.0 PL=0
MOVL C00807 V=800.0 PL=0
MOVL C00808 V=800.0 PL=0
MOVL C00809 V=800.0 PL=0
MOVL C00810 V=800.0 PL=0
MOVL C00811 V=800.0 PL=0
MOVL C00812 V=800.0 PL=0
MOVL C00813 V=800.0 PL=0
MOVL C00814 V=800.0 PL=0
MOVL C00815 V=800.0 PL=0
MOVL C00816 V=800.0 PL=0
MOVL C00817 V=800.0 PL=0
MOVL C00818 V=800.0 PL=0
MOVL C00819 V=800.0 PL=0
MOVL C00820 V=800.0 PL=0
MOVL C00821 V=800.0 PL=0
MOVL C00822 V=800.0 PL=0
MOVL C00823 V=800.0 PL=0
MOVL C00824 V=800.0 PL=0
MOVL C00825 V=800.0 PL=0
MOVL C00826 V=800.0 PL=0
MOVL C00827 V=800.0 PL=0
MOVL C00828 V=800.0 PL=0
MOVL C00829 V=800.0 PL=0
MOVL C00830 V=800.0 PL=0
MOVL C00831 V=800.0 PL=0
MOVL C00832 V=800.0 PL=0
MOVL C00833 V=800.0 PL=0
MOVL C00834 V=800.0 PL=0
MOVL C00835 V=800.0 PL=0
MOVL C00836 V=800.0 PL=0
MOVL C00837 V=800.0 PL=0
MOVL C00838 V=800.0 PL=0
MOVL C00839 V=800.0 PL=0
MOVL C00840 V=800.0 PL=0
MOVL C00841 V=800.0 PL=0
MOVL C00842 V=800.0 PL=0
MOVL C00843 V=800.0 PL=0
MOVL C00844 V=800.0 PL=0
MOVL C00845 V=800.0 PL=0
MOVL C00846 V=800.0 PL=0
MOVL C00847 V=800.0 PL=0
MOVL C00848 V=800.0 PL=0
MOVL C00849 V=800.0 PL=0
MOVL C00850 V=800.0 PL=0
MOVL C00851 V=800.0 PL=0
MOVL C00852 V=800.0 PL=0
MOVL C00853 V=800.0 PL=0
MOVL C00854 V=800.0 PL=0
MOVL C00855 V=800.0 PL=0
MOVL C00856 V=800.0 PL=0
MOVL C00857 V=800.0 PL=0
MOVL C00858 V=800.0 PL=0
MOVL C00859 V=800.0 PL=0
MOVL C00860 V=800.0 PL=0
MOVL C00861 V=800.0 PL=0
MOVL C00862 V=800.0 PL=0
MOVL C00863 V=800.0 PL=0
MOVL C00864 V=800.0 PL=0
MOVL C00865 V=800.0 PL=0
MOVL C00866 V=800.0 PL=0
MOVL C00867 V=800.0 PL=0
MOVL C00868 V=800.0 PL=0
MOVL C00869 V=800.0 PL=0
MOVL C00870 V=800.0 PL=0
MOVL C00871 V=800.0 PL=0
MOVL C00872 V=800.0 PL=0
MOVL C00873 V=800.0 PL=0
MOVL C00874 V=800.0 PL=0
MOVL C00875 V=800.0 PL=0
MOVL C00876 V=800.0 PL=0
MOVL C00877 V=800.0 PL=0
MOVL C00878 V=800.0 PL=0
MOVL C00879 V=800.0 PL=0
MOVL C00880 V=800.0 PL=0
MOVL C00881 V=800.0 PL=0
MOVL C00882 V=800.0 PL=0
MOVL C00883 V=800.0 PL=0
MOVL C00884 V=800.0 PL=0
MOVL C00885 V=800.0 PL=0
MOVL C00886 V=800.0 PL=0
MOVL C00887 V=800.0 PL=0
MOVL C00888 V=800.0 PL=0
MOVL C00889 V=800.0 PL=0
MOVL C00890 V=800.0 PL=0
MOVL C00891 V=800.0 PL=0
MOVL C00892 V=800.0 PL=0
MOVL C00893 V=800.0 PL=0
MOVL C00894 V=800.0 PL=0
MOVL C00895 V=800.0 PL=0
MOVL C00896 V=800.0 PL=0
MOVL C00897 V=800.0 PL=0
MOVL C00898 V=800.0 PL=0
MOVL C00899 V=800.0 PL=0
MOVL C00900 V=800.0 PL=0
MOVL C00901 V=800.0 PL=0
MOVL C00902 V=800.0 PL=0
MOVL C00903 V=800.0 PL=0
MOVL C00904 V=800.0 PL=0
MOVL C00905 V=800.0 PL=0
MOVL C00906 V=800.0 PL=0
MOVL C00907 V=800.0 PL=0
MOVL C00908 V=800.0 PL=0
MOVL C00909 V=800.0 PL=0
MOVL C00910 V=800.0 PL=0
MOVL C00911 V=800.0 PL=0
MOVL C00912 V=800.0 PL=0
MOVL C00913 V=800.0 PL=0
MOVL C00914 V=800.0 PL=0
MOVL C00915 V=800.0 PL=0
MOVL C00916 V=800.0 PL=0
MOVL C00917 V=800.0 PL=0
MOVL C00918 V=800.0 PL=0
MOVL C00919 V=800.0 PL=0
MOVL C00920 V=800.0 PL=0
MOVL C00921 V=800.0 PL=0
MOVL C00922 V=800.0 PL=0
MOVL C00923 V=800.0 PL=0
MOVL C00924 V=800.0 PL=0
MOVL C00925 V=800.0 PL=0
MOVL C00926 V=800.0 PL=0
MOVL C00927 V=800.0 PL=0
MOVL C00928 V=800.0 PL=0
MOVL C00929 V=800.0 PL=0
MOVL C00930 V=800.0 PL=0
MOVL C00931 V=800.0 PL=0
MOVL C00932 V=800.0 PL=0
MOVL C00933 V=800.0 PL=0
MOVL C00934 V=800.0 PL=0
MOVL C00935 V=800.0 PL=0
MOVL C00936 V=800.0 PL=0
MOVL C00937 V=800.0 PL=0
MOVL C00938 V=800.0 PL=0
MOVL C00939 V=800.0 PL=0
MOVL C00940 V=800.0 PL=0
MOVL C00941 V=800.0 PL=0
MOVL C00942 V=800.0 PL=0
MOVL C00943 V=800.0 PL=0
MOVL C00944 V=800.0 PL=0
MOVL C00945 V=800.0 PL=0
MOVL C00946 V=800.0 PL=0
MOVL C00947 V=800.0 PL=0
MOVL C00948 V=800.0 PL=0
MOVL C00949 V=800.0 PL=0
MOVL C00950 V=800.0 PL=0
MOVL C00951 V=800.0 PL=0
MOVL C00952 V=800.0 PL=0
MOVL C00953 V=800.0 PL=0
MOVL C00954 V=800.0 PL=0
MOVL C00955 V=800.0 PL=0
MOVL C00956 V=800.0 PL=0
MOVL C00957 V=800.0 PL=0
MOVL C00958 V=800.0 PL=0
MOVL C00959 V=800.0 PL=0
MOVL C00960 V=800.0 PL=0
MOVL C00961 V=800.0 PL=0
MOVL C00962 V=800.0 PL=0
MOVL C00963 V=800.0 PL=0
MOVL C00964 V=800.0 PL=0
MOVL C00965 V=800.0 PL=0
MOVL C00966 V=800.0 PL=0
MOVL C00967 V=800.0 PL=0
MOVL C00968 V=800.0 PL=0
MOVL C00969 V=800.0 PL=0
MOVL C00970 V=800.0 PL=0
MOVL C00971 V=800.0 PL=0
MOVL C00972 V=800.0 PL=0
MOVL C00973 V=800.0 PL=0
MOVL C00974 V=800.0 PL=0
MOVL C00975 V=800.0 PL=0
MOVL C00976 V=800.0 PL=0
MOVL C00977 V=800.0 PL=0
MOVL C00978 V=800.0 PL=0
MOVL C00979 V=800.0 PL=0
MOVL C00980 V=800.0 PL=0
MOVL C00981 V=800.0 PL=0
MOVL C00982 V=800.0 PL=0
MOVL C00983 V=800.0 PL=0
MOVL C00984 V=800.0 PL=0
MOVL C00985 V=800.0 PL=0
MOVL C00986 V=800.0 PL=0
MOVL C00987 V=800.0 PL=0
MOVL C00988 V=800.0 PL=0
MOVL C00989 V=800.0 PL=0
MOVL C00990 V=800.0 PL=0
MOVL C00991 V=800.0 PL=0
MOVL C00992 V=800.0 PL=0
MOVL C00993 V=800.0 PL=0
MOVL C00994 V=800.0 PL=0
MOVL C00995 V=800.0 PL=0
MOVL C00996 V=800.0 PL=0
MOVL C00997 V=800.0 PL=0
MOVL C00998 V=800.0 PL=0
MOVL C00999 V=800.0 PL=0
MOVL C01000 V=800.0 PL=0
MOVL C01001 V=800.0 PL=0
MOVL C01002 V=800.0 PL=0
MOVL C01003 V=800.0 PL=0
MOVL C01004 V=800.0 PL=0
MOVL C01005 V=800.0 PL=0
MOVL C01006 V=800.0 PL=0
MOVL C01007 V=800.0 PL=0
MOVL C01008 V=800.0 PL=0
MOVL C01009 V=800.0 PL=0
MOVL C01010 V=800.0 PL=0
MOVL C01011 V=800.0 PL=0
MOVL C01012 V=800.0 PL=0
MOVL C01013 V=800.0 PL=0
MOVL C01014 V=800.0 PL=0
MOVL C01015 V=800.0 PL=0
MOVL C01016 V=800.0 PL=0
MOVL C01017 V=800.0 PL=0
MOVL C01018 V=800.0 PL=0
MOVL C01019 V=800.0 PL=0
MOVL C01020 V=800.0 PL=0
MOVL C01021 V=800.0 PL=0
MOVL C01022 V=800.0 PL=0
MOVL C01023 V=800.0 PL=0
MOVL C01024 V=800.0 PL=0
MOVL C01025 V=800.0 PL=0
MOVL C01026 V=800.0 PL=0
MOVL C01027 V=800.0 PL=0
MOVL C01028 V=800.0 PL=0
MOVL C01029 V=800.0 PL=0
MOVL C01030 V=800.0 PL=0
MOVL C01031 V=800.0 PL=0
MOVL C01032 V=800.0 PL=0
MOVL C01033 V=800.0 PL=0
MOVL C01034 V=800.0 PL=0
MOVL C01035 V=800.0 PL=0
MOVL C01036 V=800.0 PL=0
MOVL C01037 V=800.0 PL=0
MOVL C01038 V=800.0 PL=0
MOVL C01039 V=800.0 PL=0
MOVL C01040 V=800.0 PL=0
MOVL C01041 V=800.0 PL=0
MOVL C01042 V=800.0 PL=0
MOVL C01043 V=800.0 PL=0
MOVL C01044 V=800.0 PL=0
MOVL C01045 V=800.0 PL=0
MOVL C01046 V=800.0 PL=0
MOVL C01047 V=800.0 PL=0
MOVL C01048 V=800.0 PL=0
MOVL C01049 V=800.0 PL=0
MOVL C01050 V=800.0 PL=0
MOVL C01051 V=800.0 PL=0
MOVL C01052 V=800.0 PL=0
MOVL C01053 V=800.0 PL=0
MOVL C01054 V=800.0 PL=0
MOVL C01055 V=800.0 PL=0
MOVL C01056 V=800.0 PL=0
MOVL C01057 V=800.0 PL=0
MOVL C01058 V=800.0 PL=0
MOVL C01059 V=800.0 PL=0
MOVL C01060 V=800.0 PL=0
MOVL C01061 V=800.0 PL=0
MOVL C01062 V=800.0 PL=0
MOVL C01063 V=800.0 PL=0
MOVL C01064 V=800.0 PL=0
MOVL C01065 V=800.0 PL=0
MOVL C01066 V=800.0 PL=0
MOVL C01067 V=800.0 PL=0
MOVL C01068 V=800.0 PL=0
MOVL C01069 V=800.0 PL=0
MOVL C01070 V=800.0 PL=0
MOVL C01071 V=800.0 PL=0
MOVL C01072 V=800.0 PL=0
MOVL C01073 V=800.0 PL=0
MOVL C01074 V=800.0 PL=0
MOVL C01075 V=800.0 PL=0
MOVL C01076 V=800.0 PL=0
MOVL C01077 V=800.0 PL=0
MOVL C01078 V=800.0 PL=0
MOVL C01079 V=800.0 PL=0
MOVL C01080 V=800.0 PL=0
MOVL C01081 V=800.0 PL=0
MOVL C01082 V=800.0 PL=0
MOVL C01083 V=800.0 PL=0
MOVL C01084 V=800.0 PL=0
MOVL C01085 V=800.0 PL=0
MOVL C01086 V=800.0 PL=0
MOVL C01087 V=800.0 PL=0
MOVL C01088 V=800.0 PL=0
MOVL C01089 V=800.0 PL=0
MOVL C01090 V=800.0 PL=0
MOVL C01091 V=800.0 PL=0
MOVL C01092 V=800.0 PL=0
MOVL C01093 V=800.0 PL=0
MOVL C01094 V=800.0 PL=0
MOVL C01095 V=800.0 PL=0
MOVL C01096 V=800.0 PL=0
MOVL C01097 V=800.0 PL=0
MOVL C01098 V=800.0 PL=0
MOVL C01099 V=800.0 PL=0
MOVL C01100 V=800.0 PL=0
MOVL C01101 V=800.0 PL=0
MOVL C01102 V=800.0 PL=0
MOVL C01103 V=800.0 PL=0
MOVL C01104 V=800.0 PL=0
MOVL C01105 V=800.0 PL=0
MOVL C01106 V=800.0 PL=0
MOVL C01107 V=800.0 PL=0
MOVL C01108 V=800.0 PL=0
MOVL C01109 V=800.0 PL=0
MOVL C01110 V=800.0 PL=0
MOVL C01111 V=800.0 PL=0
MOVL C01112 V=800.0 PL=0
MOVL C01113 V=800.0 PL=0
MOVL C01114 V=800.0 PL=0
MOVL C01115 V=800.0 PL=0
MOVL C01116 V=800.0 PL=0
MOVL C01117 V=800.0 PL=0
MOVL C01118 V=800.0 PL=0
MOVL C01119 V=800.0 PL=0
MOVL C01120 V=800.0 PL=0
MOVL C01121 V=800.0 PL=0
MOVL C01122 V=800.0 PL=0
MOVL C01123 V=800.0 PL=0
MOVL C01124 V=800.0 PL=0
MOVL C01125 V=800.0 PL=0
MOVL C01126 V=800.0 PL=0
MOVL C01127 V=800.0 PL=0
MOVL C01128 V=800.0 PL=0
MOVL C01129 V=800.0 PL=0
MOVL C01130 V=800.0 PL=0
MOVL C01131 V=800.0 PL=0
MOVL C01132 V=800.0 PL=0
MOVL C01133 V=800.0 PL=0
MOVL C01134 V=800.0 PL=0
MOVL C01135 V=800.0 PL=0
MOVL C01136 V=800.0 PL=0
MOVL C01137 V=800.0 PL=0
MOVL C01138 V=800.0 PL=0
MOVL C01139 V=800.0 PL=0
MOVL C01140 V=800.0 PL=0
MOVL C01141 V=800.0 PL=0
MOVL C01142 V=800.0 PL=0
MOVL C01143 V=800.0 PL=0
MOVL C01144 V=800.0 PL=0
MOVL C01145 V=800.0 PL=0
MOVL C01146 V=800.0 PL=0
MOVL C01147 V=800.0 PL=0
MOVL C01148 V=800.0 PL=0
MOVL C01149 V=800.0 PL=0
MOVL C01150 V=800.0 PL=0
MOVL C01151 V=800.0 PL=0
MOVL C01152 V=800.0 PL=0
MOVL C01153 V=800.0 PL=0
MOVL C01154 V=800.0 PL=0
MOVL C01155 V=800.0 PL=0
MOVL C01156 V=800.0 PL=0
MOVL C01157 V=800.0 PL=0
MOVL C01158 V=800.0 PL=0
MOVL C01159 V=800.0 PL=0
MOVL C01160 V=800.0 PL=0
MOVL C01161 V=800.0 PL=0
MOVL C01162 V=800.0 PL=0
MOVL C01163 V=800.0 PL=0
MOVL C01164 V=800.0 PL=0
MOVL C01165 V=800.0 PL=0
MOVL C01166 V=800.0 PL=0
MOVL C01167 V=800.0 PL=0
MOVL C01168 V=800.0 PL=0
MOVL C01169 V=800.0 PL=0
MOVL C01170 V=800.0 PL=0
MOVL C01171 V=800.0 PL=0
MOVL C01172 V=800.0 PL=0
MOVL C01173 V=800.0 PL=0
MOVL C01174 V=800.0 PL=0
MOVL C01175 V=800.0 PL=0
MOVL C01176 V=800.0 PL=0
MOVL C01177 V=800.0 PL=0
MOVL C01178 V=800.0 PL=0
MOVL C01179 V=800.0 PL=0
MOVL C01180 V=800.0 PL=0
MOVL C01181 V=800.0 PL=0
MOVL C01182 V=800.0 PL=0
MOVL C01183 V=800.0 PL=0
MOVL C01184 V=800.0 PL=0
MOVL C01185 V=800.0 PL=0
MOVL C01186 V=800.0 PL=0
MOVL C01187 V=800.0 PL=0
MOVL C01188 V=800.0 PL=0
MOVL C01189 V=800.0 PL=0
MOVL C01190 V=800.0 PL=0
MOVL C01191 V=800.0 PL=0
MOVL C01192 V=800.0 PL=0
MOVL C01193 V=800.0 PL=0
MOVL C01194 V=800.0 PL=0
MOVL C01195 V=800.0 PL=0
MOVL C01196 V=800.0 PL=0
MOVL C01197 V=800.0 PL=0
MOVL C01198 V=800.0 PL=0
MOVL C01199 V=800.0 PL=0
MOVL C01200 V=800.0 PL=0
MOVL C01201 V=800.0 PL=0
MOVL C01202 V=800.0 PL=0
MOVL C01203 V=800.0 PL=0
MOVL C01204 V=800.0 PL=0
MOVL C01205 V=800.0 PL=0
MOVL C01206 V=800.0 PL=0
MOVL C01207 V=800.0 PL=0
MOVL C01208 V=800.0 PL=0
MOVL C01209 V=800.0 PL=0
MOVL C01210 V=800.0 PL=0
MOVL C01211 V=800.0 PL=0
MOVL C01212 V=800.0 PL=0
MOVL C01213 V=800.0 PL=0
MOVL C01214 V=800.0 PL=0
MOVL C01215 V=800.0 PL=0
MOVL C01216 V=800.0 PL=0
MOVL C01217 V=800.0 PL=0
MOVL C01218 V=800.0 PL=0
MOVL C01219 V=800.0 PL=0
MOVL C01220 V=800.0 PL=0
MOVL C01221 V=800.0 PL=0
MOVL C01222 V=800.0 PL=0
MOVL C01223 V=800.0 PL=0
MOVL C01224 V=800.0 PL=0
MOVL C01225 V=800.0 PL=0
MOVL C01226 V=800.0 PL=0
MOVL C01227 V=800.0 PL=0
MOVL C01228 V=800.0 PL=0
MOVL C01229 V=800.0 PL=0
MOVL C01230 V=800.0 PL=0
MOVL C01231 V=800.0 PL=0
MOVL C01232 V=800.0 PL=0
MOVL C01233 V=800.0 PL=0
MOVL C01234 V=800.0 PL=0
MOVL C01235 V=800.0 PL=0
MOVL C01236 V=800.0 PL=0
MOVL C01237 V=800.0 PL=0
MOVL C01238 V=800.0 PL=0
MOVL C01239 V=800.0 PL=0
MOVL C01240 V=800.0 PL=0
MOVL C01241 V=800.0 PL=0
MOVL C01242 V=800.0 PL=0
MOVL C01243 V=800.0 PL=0
MOVL C01244 V=800.0 PL=0
MOVL C01245 V=800.0 PL=0
MOVL C01246 V=800.0 PL=0
MOVL C01247 V=800.0 PL=0
MOVL C01248 V=800.0 PL=0
MOVL C01249 V=800.0 PL=0
MOVL C01250 V=800.0 PL=0
MOVL C01251 V=800.0 PL=0
MOVL C01252 V=800.0 PL=0
MOVL C01253 V=800.0 PL=0
MOVL C01254 V=800.0 PL=0
MOVL C01255 V=800.0 PL=0
MOVL C01256 V=800.0 PL=0
MOVL C01257 V=800.0 PL=0
MOVL C01258 V=800.0 PL=0
MOVL C01259 V=800.0 PL=0
MOVL C01260 V=800.0 PL=0
MOVL C01261 V=800.0 PL=0
MOVL C01262 V=800.0 PL=0
MOVL C01263 V=800.0 PL=0
MOVL C01264 V=800.0 PL=0
MOVL C01265 V=800.0 PL=0
MOVL C01266 V=800.0 PL=0
MOVL C01267 V=800.0 PL=0
MOVL C01268 V=800.0 PL=0
MOVL C01269 V=800.0 PL=0
MOVL C01270 V=800.0 PL=0
MOVL C01271 V=800.0 PL=0
MOVL C01272 V=800.0 PL=0
MOVL C01273 V=800.0 PL=0
MOVL C01274 V=800.0 PL=0
MOVL C01275 V=800.0 PL=0
MOVL C01276 V=800.0 PL=0
MOVL C01277 V=800.0 PL=0
MOVL C01278 V=800.0 PL=0
MOVL C01279 V=800.0 PL=0
MOVL C01280 V=800.0 PL=0
MOVL C01281 V=800.0 PL=0
MOVL C01282 V=800.0 PL=0
MOVL C01283 V=800.0 PL=0
MOVL C01284 V=800.0 PL=0
MOVL C01285 V=800.0 PL=0
MOVL C01286 V=800.0 PL=0
MOVL C01287 V=800.0 PL=0
MOVL C01288 V=800.0 PL=0
MOVL C01289 V=800.0 PL=0
MOVL C01290 V=800.0 PL=0
MOVL C01291 V=800.0 PL=0
MOVL C01292 V=800.0 PL=0
MOVL C01293 V=800.0 PL=0
MOVL C01294 V=800.0 PL=0
MOVL C01295 V=800.0 PL=0
MOVL C01296 V=800.0 PL=0
MOVL C01297 V=800.0 PL=0
MOVL C01298 V=800.0 PL=0
MOVL C01299 V=800.0 PL=0
MOVL C01300 V=800.0 PL=0
MOVL C01301 V=800.0 PL=0
MOVL C01302 V=800.0 PL=0
MOVL C01303 V=800.0 PL=0
MOVL C01304 V=800.0 PL=0
MOVL C01305 V=800.0 PL=0
MOVL C01306 V=800.0 PL=0
MOVL C01307 V=800.0 PL=0
MOVL C01308 V=800.0 PL=0
MOVL C01309 V=800.0 PL=0
MOVL C01310 V=800.0 PL=0
MOVL C01311 V=800.0 PL=0
MOVL C01312 V=800.0 PL=0
MOVL C01313 V=800.0 PL=0
MOVL C01314 V=800.0 PL=0
MOVL C01315 V=800.0 PL=0
MOVL C01316 V=800.0 PL=0
MOVL C01317 V=800.0 PL=0
MOVL C01318 V=800.0 PL=0
MOVL C01319 V=800.0 PL=0
MOVL C01320 V=800.0 PL=0
MOVL C01321 V=800.0 PL=0
MOVL C01322 V=800.0 PL=0
MOVL C01323 V=800.0 PL=0
MOVL C01324 V=800.0 PL=0
MOVL C01325 V=800.0 PL=0
MOVL C01326 V=800.0 PL=0
MOVL C01327 V=800.0 PL=0
MOVL C01328 V=800.0 PL=0
MOVL C01329 V=800.0 PL=0
MOVL C01330 V=800.0 PL=0
MOVL C01331 V=800.0 PL=0
MOVL C01332 V=800.0 PL=0
MOVL C01333 V=800.0 PL=0
MOVL C01334 V=800.0 PL=0
MOVL C01335 V=800.0 PL=0
MOVL C01336 V=800.0 PL=0
MOVL C01337 V=800.0 PL=0
MOVL C01338 V=800.0 PL=0
MOVL C01339 V=800.0 PL=0
MOVL C01340 V=800.0 PL=0
MOVL C01341 V=800.0 PL=0
MOVL C01342 V=800.0 PL=0
MOVL C01343 V=800.0 PL=0
MOVL C01344 V=800.0 PL=0
MOVL C01345 V=800.0 PL=0
MOVL C01346 V=800.0 PL=0
MOVL C01347 V=800.0 PL=0
MOVL C01348 V=800.0 PL=0
MOVL C01349 V=800.0 PL=0
MOVL C01350 V=800.0 PL=0
MOVL C01351 V=800.0 PL=0
MOVL C01352 V=800.0 PL=0
MOVL C01353 V=800.0 PL=0
MOVL C01354 V=800.0 PL=0
MOVL C01355 V=800.0 PL=0
MOVL C01356 V=800.0 PL=0
MOVL C01357 V=800.0 PL=0
MOVL C01358 V=800.0 PL=0
MOVL C01359 V=800.0 PL=0
MOVL C01360 V=800.0 PL=0
MOVL C01361 V=800.0 PL=0
MOVL C01362 V=800.0 PL=0
MOVL C01363 V=800.0 PL=0
MOVL C01364 V=800.0 PL=0
MOVL C01365 V=800.0 PL=0
MOVL C01366 V=800.0 PL=0
MOVL C01367 V=800.0 PL=0
MOVL C01368 V=800.0 PL=0
MOVL C01369 V=800.0 PL=0
MOVL C01370 V=800.0 PL=0
MOVL C01371 V=800.0 PL=0
MOVL C01372 V=800.0 PL=0
MOVL C01373 V=800.0 PL=0
MOVL C01374 V=800.0 PL=0
MOVL C01375 V=800.0 PL=0
MOVL C01376 V=800.0 PL=0
MOVL C01377 V=800.0 PL=0
MOVL C01378 V=800.0 PL=0
MOVL C01379 V=800.0 PL=0
MOVL C01380 V=800.0 PL=0
MOVL C01381 V=800.0 PL=0
MOVL C01382 V=800.0 PL=0
MOVL C01383 V=800.0 PL=0
MOVL C01384 V=800.0 PL=0
MOVL C01385 V=800.0 PL=0
MOVL C01386 V=800.0 PL=0
MOVL C01387 V=800.0 PL=0
MOVL C01388 V=800.0 PL=0
MOVL C01389 V=800.0 PL=0
MOVL C01390 V=800.0 PL=0
MOVL C01391 V=800.0 PL=0
MOVL C01392 V=800.0 PL=0
MOVL C01393 V=800.0 PL=0
MOVL C01394 V=800.0 PL=0
MOVL C01395 V=800.0 PL=0
MOVL C01396 V=800.0 PL=0
MOVL C01397 V=800.0 PL=0
MOVL C01398 V=800.0 PL=0
MOVL C01399 V=800.0 PL=0
MOVL C01400 V=800.0 PL=0
MOVL C01401 V=800.0 PL=0
MOVL C01402 V=800.0 PL=0
MOVL C01403 V=800.0 PL=0
MOVL C01404 V=800.0 PL=0
MOVL C01405 V=800.0 PL=0
MOVL C01406 V=800.0 PL=0
MOVL C01407 V=800.0 PL=0
MOVL C01408 V=800.0 PL=0
MOVL C01409 V=800.0 PL=0
MOVL C01410 V=800.0 PL=0
MOVL C01411 V=800.0 PL=0
MOVL C01412 V=800.0 PL=0
MOVL C01413 V=800.0 PL=0
MOVL C01414 V=800.0 PL=0
MOVL C01415 V=800.0 PL=0
MOVL C01416 V=800.0 PL=0
MOVL C01417 V=800.0 PL=0
MOVL C01418 V=800.0 PL=0
MOVL C01419 V=800.0 PL=0
MOVL C01420 V=800.0 PL=0
MOVL C01421 V=800.0 PL=0
MOVL C01422 V=800.0 PL=0
MOVL C01423 V=800.0 PL=0
MOVL C01424 V=800.0 PL=0
MOVL C01425 V=800.0 PL=0
MOVL C01426 V=800.0 PL=0
MOVL C01427 V=800.0 PL=0
MOVL C01428 V=800.0 PL=0
MOVL C01429 V=800.0 PL=0
MOVL C01430 V=800.0 PL=0
MOVL C01431 V=800.0 PL=0
MOVL C01432 V=800.0 PL=0
MOVL C01433 V=800.0 PL=0
MOVL C01434 V=800.0 PL=0
MOVL C01435 V=800.0 PL=0
MOVL C01436 V=800.0 PL=0
MOVL C01437 V=800.0 PL=0
MOVL C01438 V=800.0 PL=0
MOVL C01439 V=800.0 PL=0
MOVL C01440 V=800.0 PL=0
MOVL C01441 V=800.0 PL=0
MOVL C01442 V=800.0 PL=0
MOVL C01443 V=800.0 PL=0
MOVL C01444 V=800.0 PL=0
MOVL C01445 V=800.0 PL=0
MOVL C01446 V=800.0 PL=0
MOVL C01447 V=800.0 PL=0
MOVL C01448 V=800.0 PL=0
MOVL C01449 V=800.0 PL=0
MOVL C01450 V=800.0 PL=0
MOVL C01451 V=800.0 PL=0
MOVL C01452 V=800.0 PL=0
MOVL C01453 V=800.0 PL=0
MOVL C01454 V=800.0 PL=0
MOVL C01455 V=800.0 PL=0
MOVL C01456 V=800.0 PL=0
MOVL C01457 V=800.0 PL=0
MOVL C01458 V=800.0 PL=0
MOVL C01459 V=800.0 PL=0
MOVL C01460 V=800.0 PL=0
MOVL C01461 V=800.0 PL=0
MOVL C01462 V=800.0 PL=0
MOVL C01463 V=800.0 PL=0
MOVL C01464 V=800.0 PL=0
MOVL C01465 V=800.0 PL=0
MOVL C01466 V=800.0 PL=0
MOVL C01467 V=800.0 PL=0
MOVL C01468 V=800.0 PL=0
MOVL C01469 V=800.0 PL=0
MOVL C01470 V=800.0 PL=0
MOVL C01471 V=800.0 PL=0
MOVL C01472 V=800.0 PL=0
MOVL C01473 V=800.0 PL=0
MOVL C01474 V=800.0 PL=0
MOVL C01475 V=800.0 PL=0
MOVL C01476 V=800.0 PL=0
MOVL C01477 V=800.0 PL=0
MOVL C01478 V=800.0 PL=0
MOVL C01479 V=800.0 PL=0
MOVL C01480 V=800.0 PL=0
MOVL C01481 V=800.0 PL=0
MOVL C01482 V=800.0 PL=0
MOVL C01483 V=800.0 PL=0
MOVL C01484 V=800.0 PL=0
MOVL C01485 V=800.0 PL=0
MOVL C01486 V=800.0 PL=0
MOVL C01487 V=800.0 PL=0
MOVL C01488 V=800.0 PL=0
MOVL C01489 V=800.0 PL=0
MOVL C01490 V=800.0 PL=0
MOVL C01491 V=800.0 PL=0
MOVL C01492 V=800.0 PL=0
MOVL C01493 V=800.0 PL=0
MOVL C01494 V=800.0 PL=0
MOVL C01495 V=800.0 PL=0
MOVL C01496 V=800.0 PL=0
MOVL C01497 V=800.0 PL=0
MOVL C01498 V=800.0 PL=0
MOVL C01499 V=800.0 PL=0
MOVL C01500 V=800.0 PL=0
MOVL C01501 V=800.0 PL=0
MOVL C01502 V=800.0 PL=0
MOVL C01503 V=800.0 PL=0
MOVL C01504 V=800.0 PL=0
MOVL C01505 V=800.0 PL=0
MOVL C01506 V=800.0 PL=0
MOVL C01507 V=800.0 PL=0
MOVL C01508 V=800.0 PL=0
MOVL C01509 V=800.0 PL=0
MOVL C01510 V=800.0 PL=0
MOVL C01511 V=800.0 PL=0
MOVL C01512 V=800.0 PL=0
MOVL C01513 V=800.0 PL=0
MOVL C01514 V=800.0 PL=0
MOVL C01515 V=800.0 PL=0
MOVL C01516 V=800.0 PL=0
MOVL C01517 V=800.0 PL=0
MOVL C01518 V=800.0 PL=0
MOVL C01519 V=800.0 PL=0
MOVL C01520 V=800.0 PL=0
MOVL C01521 V=800.0 PL=0
MOVL C01522 V=800.0 PL=0
MOVL C01523 V=800.0 PL=0
MOVL C01524 V=800.0 PL=0
MOVL C01525 V=800.0 PL=0
MOVL C01526 V=800.0 PL=0
MOVL C01527 V=800.0 PL=0
MOVL C01528 V=800.0 PL=0
MOVL C01529 V=800.0 PL=0
MOVL C01530 V=800.0 PL=0
MOVL C01531 V=800.0 PL=0
MOVL C01532 V=800.0 PL=0
MOVL C01533 V=800.0 PL=0
MOVL C01534 V=800.0 PL=0
MOVL C01535 V=800.0 PL=0
MOVL C01536 V=800.0 PL=0
MOVL C01537 V=800.0 PL=0
MOVL C01538 V=800.0 PL=0
MOVL C01539 V=800.0 PL=0
MOVL C01540 V=800.0 PL=0
MOVL C01541 V=800.0 PL=0
MOVL C01542 V=800.0 PL=0
MOVL C01543 V=800.0 PL=0
MOVL C01544 V=800.0 PL=0
MOVL C01545 V=800.0 PL=0
MOVL C01546 V=800.0 PL=0
MOVL C01547 V=800.0 PL=0
MOVL C01548 V=800.0 PL=0
MOVL C01549 V=800.0 PL=0
MOVL C01550 V=800.0 PL=0
MOVL C01551 V=800.0 PL=0
MOVL C01552 V=800.0 PL=0
MOVL C01553 V=800.0 PL=0
MOVL C01554 V=800.0 PL=0
MOVL C01555 V=800.0 PL=0
MOVL C01556 V=800.0 PL=0
MOVL C01557 V=800.0 PL=0
MOVL C01558 V=800.0 PL=0
MOVL C01559 V=800.0 PL=0
MOVL C01560 V=800.0 PL=0
MOVL C01561 V=800.0 PL=0
MOVL C01562 V=800.0 PL=0
MOVL C01563 V=800.0 PL=0
MOVL C01564 V=800.0 PL=0
MOVL C01565 V=800.0 PL=0
MOVL C01566 V=800.0 PL=0
MOVL C01567 V=800.0 PL=0
MOVL C01568 V=800.0 PL=0
MOVL C01569 V=800.0 PL=0
MOVL C01570 V=800.0 PL=0
MOVL C01571 V=800.0 PL=0
MOVL C01572 V=800.0 PL=0
MOVL C01573 V=800.0 PL=0
MOVL C01574 V=800.0 PL=0
MOVL C01575 V=800.0 PL=0
MOVL C01576 V=800.0 PL=0
MOVL C01577 V=800.0 PL=0
MOVL C01578 V=800.0 PL=0
MOVL C01579 V=800.0 PL=0
MOVL C01580 V=800.0 PL=0
MOVL C01581 V=800.0 PL=0
MOVL C01582 V=800.0 PL=0
MOVL C01583 V=800.0 PL=0
MOVL C01584 V=800.0 PL=0
MOVL C01585 V=800.0 PL=0
MOVL C01586 V=800.0 PL=0
MOVL C01587 V=800.0 PL=0
MOVL C01588 V=800.0 PL=0
MOVL C01589 V=800.0 PL=0
MOVL C01590 V=800.0 PL=0
MOVL C01591 V=800.0 PL=0
MOVL C01592 V=800.0 PL=0
MOVL C01593 V=800.0 PL=0
MOVL C01594 V=800.0 PL=0
MOVL C01595 V=800.0 PL=0
MOVL C01596 V=800.0 PL=0
MOVL C01597 V=800.0 PL=0
MOVL C01598 V=800.0 PL=0
MOVL C01599 V=800.0 PL=0
MOVL C01600 V=800.0 PL=0
MOVL C01601 V=800.0 PL=0
MOVL C01602 V=800.0 PL=0
MOVL C01603 V=800.0 PL=0
MOVL C01604 V=800.0 PL=0
MOVL C01605 V=800.0 PL=0
MOVL C01606 V=800.0 PL=0
MOVL C01607 V=800.0 PL=0
MOVL C01608 V=800.0 PL=0
MOVL C01609 V=800.0 PL=0
MOVL C01610 V=800.0 PL=0
MOVL C01611 V=800.0 PL=0
MOVL C01612 V=800.0 PL=0
MOVL C01613 V=800.0 PL=0
MOVL C01614 V=800.0 PL=0
MOVL C01615 V=800.0 PL=0
MOVL C01616 V=800.0 PL=0
MOVL C01617 V=800.0 PL=0
MOVL C01618 V=800.0 PL=0
MOVL C01619 V=800.0 PL=0
MOVL C01620 V=800.0 PL=0
MOVL C01621 V=800.0 PL=0
MOVL C01622 V=800.0 PL=0
MOVL C01623 V=800.0 PL=0
MOVL C01624 V=800.0 PL=0
MOVL C01625 V=800.0 PL=0
MOVL C01626 V=800.0 PL=0
MOVL C01627 V=800.0 PL=0
MOVL C01628 V=800.0 PL=0
MOVL C01629 V=800.0 PL=0
MOVL C01630 V=800.0 PL=0
MOVL C01631 V=800.0 PL=0
MOVL C01632 V=800.0 PL=0
MOVL C01633 V=800.0 PL=0
MOVL C01634 V=800.0 PL=0
MOVL C01635 V=800.0 PL=0
MOVL C01636 V=800.0 PL=0
MOVL C01637 V=800.0 PL=0
MOVL C01638 V=800.0 PL=0
MOVL C01639 V=800.0 PL=0
MOVL C01640 V=800.0 PL=0
MOVL C01641 V=800.0 PL=0
MOVL C01642 V=800.0 PL=0
MOVL C01643 V=800.0 PL=0
MOVL C01644 V=800.0 PL=0
MOVL C01645 V=800.0 PL=0
MOVL C01646 V=800.0 PL=0
MOVL C01647 V=800.0 PL=0
MOVL C01648 V=800.0 PL=0
MOVL C01649 V=800.0 PL=0
MOVL C01650 V=800.0 PL=0
MOVL C01651 V=800.0 PL=0
MOVL C01652 V=800.0 PL=0
MOVL C01653 V=800.0 PL=0
MOVL C01654 V=800.0 PL=0
MOVL C01655 V=800.0 PL=0
MOVL C01656 V=800.0 PL=0
MOVL C01657 V=800.0 PL=0
MOVL C01658 V=800.0 PL=0
MOVL C01659 V=800.0 PL=0
MOVL C01660 V=800.0 PL=0
MOVL C01661 V=800.0 PL=0
MOVL C01662 V=800.0 PL=0
MOVL C01663 V=800.0 PL=0
MOVL C01664 V=800.0 PL=0
MOVL C01665 V=800.0 PL=0
MOVL C01666 V=800.0 PL=0
MOVL C01667 V=800.0 PL=0
MOVL C01668 V=800.0 PL=0
MOVL C01669 V=800.0 PL=0
MOVL C01670 V=800.0 PL=0
MOVL C01671 V=800.0 PL=0
MOVL C01672 V=800.0 PL=0
MOVL C01673 V=800.0 PL=0
MOVL C01674 V=800.0 PL=0
MOVL C01675 V=800.0 PL=0
MOVL C01676 V=800.0 PL=0
MOVL C01677 V=800.0 PL=0
MOVL C01678 V=800.0 PL=0
MOVL C01679 V=800.0 PL=0
MOVL C01680 V=800.0 PL=0
MOVL C01681 V=800.0 PL=0
MOVL C01682 V=800.0 PL=0
MOVL C01683 V=800.0 PL=0
MOVL C01684 V=800.0 PL=0
MOVL C01685 V=800.0 PL=0
MOVL C01686 V=800.0 PL=0
MOVL C01687 V=800.0 PL=0
MOVL C01688 V=800.0 PL=0
MOVL C01689 V=800.0 PL=0
MOVL C01690 V=800.0 PL=0
MOVL C01691 V=800.0 PL=0
MOVL C01692 V=800.0 PL=0
MOVL C01693 V=800.0 PL=0
MOVL C01694 V=800.0 PL=0
MOVL C01695 V=800.0 PL=0
MOVL C01696 V=800.0 PL=0
MOVL C01697 V=800.0 PL=0
MOVL C01698 V=800.0 PL=0
MOVL C01699 V=800.0 PL=0
MOVL C01700 V=800.0 PL=0
MOVL C01701 V=800.0 PL=0
MOVL C01702 V=800.0 PL=0
MOVL C01703 V=800.0 PL=0
MOVL C01704 V=800.0 PL=0
MOVL C01705 V=800.0 PL=0
MOVL C01706 V=800.0 PL=0
MOVL C01707 V=800.0 PL=0
MOVL C01708 V=800.0 PL=0
MOVL C01709 V=800.0 PL=0
MOVL C01710 V=800.0 PL=0
MOVL C01711 V=800.0 PL=0
MOVL C01712 V=800.0 PL=0
MOVL C01713 V=800.0 PL=0
MOVL C01714 V=800.0 PL=0
MOVL C01715 V=800.0 PL=0
MOVL C01716 V=800.0 PL=0
MOVL C01717 V=800.0 PL=0
MOVL C01718 V=800.0 PL=0
MOVL C01719 V=800.0 PL=0
MOVL C01720 V=800.0 PL=0
MOVL C01721 V=800.0 PL=0
MOVL C01722 V=800.0 PL=0
MOVL C01723 V=800.0 PL=0
MOVL C01724 V=800.0 PL=0
MOVL C01725 V=800.0 PL=0
MOVL C01726 V=800.0 PL=0
MOVL C01727 V=800.0 PL=0
MOVL C01728 V=800.0 PL=0
MOVL C01729 V=800.0 PL=0
MOVL C01730 V=800.0 PL=0
MOVL C01731 V=800.0 PL=0
MOVL C01732 V=800.0 PL=0
MOVL C01733 V=800.0 PL=0
MOVL C01734 V=800.0 PL=0
MOVL C01735 V=800.0 PL=0
MOVL C01736 V=800.0 PL=0
MOVL C01737 V=800.0 PL=0
MOVL C01738 V=800.0 PL=0
MOVL C01739 V=800.0 PL=0
MOVL C01740 V=800.0 PL=0
MOVL C01741 V=800.0 PL=0
MOVL C01742 V=800.0 PL=0
MOVL C01743 V=800.0 PL=0
MOVL C01744 V=800.0 PL=0
MOVL C01745 V=800.0 PL=0
MOVL C01746 V=800.0 PL=0
MOVL C01747 V=800.0 PL=0
MOVL C01748 V=800.0 PL=0
MOVL C01749 V=800.0 PL=0
MOVL C01750 V=800.0 PL=0
MOVL C01751 V=800.0 PL=0
MOVL C01752 V=800.0 PL=0
MOVL C01753 V=800.0 PL=0
MOVL C01754 V=800.0 PL=0
MOVL C01755 V=800.0 PL=0
MOVL C01756 V=800.0 PL=0
MOVL C01757 V=800.0 PL=0
MOVL C01758 V=800.0 PL=0
MOVL C01759 V=800.0 PL=0
MOVL C01760 V=800.0 PL=0
MOVL C01761 V=800.0 PL=0
MOVL C01762 V=800.0 PL=0
MOVL C01763 V=800.0 PL=0
MOVL C01764 V=800.0 PL=0
MOVL C01765 V=800.0 PL=0
MOVL C01766 V=800.0 PL=0
MOVL C01767 V=800.0 PL=0
MOVL C01768 V=800.0 PL=0
MOVL C01769 V=800.0 PL=0
MOVL C01770 V=800.0 PL=0
MOVL C01771 V=800.0 PL=0
MOVL C01772 V=800.0 PL=0
MOVL C01773 V=800.0 PL=0
MOVL C01774 V=800.0 PL=0
MOVL C01775 V=800.0 PL=0
MOVL C01776 V=800.0 PL=0
MOVL C01777 V=800.0 PL=0
MOVL C01778 V=800.0 PL=0
MOVL C01779 V=800.0 PL=0
MOVL C01780 V=800.0 PL=0
MOVL C01781 V=800.0 PL=0
MOVL C01782 V=800.0 PL=0
MOVL C01783 V=800.0 PL=0
MOVL C01784 V=800.0 PL=0
MOVL C01785 V=800.0 PL=0
MOVL C01786 V=800.0 PL=0
MOVL C01787 V=800.0 PL=0
MOVL C01788 V=800.0 PL=0
MOVL C01789 V=800.0 PL=0
MOVL C01790 V=800.0 PL=0
MOVL C01791 V=800.0 PL=0
MOVL C01792 V=800.0 PL=0
MOVL C01793 V=800.0 PL=0
MOVL C01794 V=800.0 PL=0
MOVL C01795 V=800.0 PL=0
MOVL C01796 V=800.0 PL=0
MOVL C01797 V=800.0 PL=0
MOVL C01798 V=800.0 PL=0
MOVL C01799 V=800.0 PL=0
MOVL C01800 V=800.0 PL=0
MOVL C01801 V=800.0 PL=0
MOVL C01802 V=800.0 PL=0
MOVL C01803 V=800.0 PL=0
MOVL C01804 V=800.0 PL=0
MOVL C01805 V=800.0 PL=0
MOVL C01806 V=800.0 PL=0
MOVL C01807 V=800.0 PL=0
MOVL C01808 V=800.0 PL=0
MOVL C01809 V=800.0 PL=0
MOVL C01810 V=800.0 PL=0
MOVL C01811 V=800.0 PL=0
MOVL C01812 V=800.0 PL=0
MOVL C01813 V=800.0 PL=0
MOVL C01814 V=800.0 PL=0
MOVL C01815 V=800.0 PL=0
MOVL C01816 V=800.0 PL=0
MOVL C01817 V=800.0 PL=0
MOVL C01818 V=800.0 PL=0
MOVL C01819 V=800.0 PL=0
MOVL C01820 V=800.0 PL=0
MOVL C01821 V=800.0 PL=0
MOVL C01822 V=800.0 PL=0
MOVL C01823 V=800.0 PL=0
MOVL C01824 V=800.0 PL=0
MOVL C01825 V=800.0 PL=0
MOVL C01826 V=800.0 PL=0
MOVL C01827 V=800.0 PL=0
MOVL C01828 V=800.0 PL=0
MOVL C01829 V=800.0 PL=0
MOVL C01830 V=800.0 PL=0
MOVL C01831 V=800.0 PL=0
MOVL C01832 V=800.0 PL=0
MOVL C01833 V=800.0 PL=0
MOVL C01834 V=800.0 PL=0
MOVL C01835 V=800.0 PL=0
MOVL C01836 V=800.0 PL=0
MOVL C01837 V=800.0 PL=0
MOVL C01838 V=800.0 PL=0
MOVL C01839 V=800.0 PL=0
MOVL C01840 V=800.0 PL=0
MOVL C01841 V=800.0 PL=0
MOVL C01842 V=800.0 PL=0
MOVL C01843 V=800.0 PL=0
MOVL C01844 V=800.0 PL=0
MOVL C01845 V=800.0 PL=0
MOVL C01846 V=800.0 PL=0
MOVL C01847 V=800.0 PL=0
MOVL C01848 V=800.0 PL=0
MOVL C01849 V=800.0 PL=0
MOVL C01850 V=800.0 PL=0
MOVL C01851 V=800.0 PL=0
MOVL C01852 V=800.0 PL=0
MOVL C01853 V=800.0 PL=0
MOVL C01854 V=800.0 PL=0
MOVL C01855 V=800.0 PL=0
MOVL C01856 V=800.0 PL=0
MOVL C01857 V=800.0 PL=0
MOVL C01858 V=800.0 PL=0
MOVL C01859 V=800.0 PL=0
MOVL C01860 V=800.0 PL=0
MOVL C01861 V=800.0 PL=0
MOVL C01862 V=800.0 PL=0
MOVL C01863 V=800.0 PL=0
MOVL C01864 V=800.0 PL=0
MOVL C01865 V=800.0 PL=0
MOVL C01866 V=800.0 PL=0
MOVL C01867 V=800.0 PL=0
MOVL C01868 V=800.0 PL=0
MOVL C01869 V=800.0 PL=0
MOVL C01870 V=800.0 PL=0
MOVL C01871 V=800.0 PL=0
MOVL C01872 V=800.0 PL=0
MOVL C01873 V=800.0 PL=0
MOVL C01874 V=800.0 PL=0
MOVL C01875 V=800.0 PL=0
MOVL C01876 V=800.0 PL=0
MOVL C01877 V=800.0 PL=0
MOVL C01878 V=800.0 PL=0
MOVL C01879 V=800.0 PL=0
MOVL C01880 V=800.0 PL=0
MOVL C01881 V=800.0 PL=0
MOVL C01882 V=800.0 PL=0
MOVL C01883 V=800.0 PL=0
MOVL C01884 V=800.0 PL=0
MOVL C01885 V=800.0 PL=0
MOVL C01886 V=800.0 PL=0
MOVL C01887 V=800.0 PL=0
MOVL C01888 V=800.0 PL=0
MOVL C01889 V=800.0 PL=0
MOVL C01890 V=800.0 PL=0
MOVL C01891 V=800.0 PL=0
MOVL C01892 V=800.0 PL=0
MOVL C01893 V=800.0 PL=0
MOVL C01894 V=800.0 PL=0
MOVL C01895 V=800.0 PL=0
MOVL C01896 V=800.0 PL=0
MOVL C01897 V=800.0 PL=0
MOVL C01898 V=800.0 PL=0
MOVL C01899 V=800.0 PL=0
MOVL C01900 V=800.0 PL=0
MOVL C01901 V=800.0 PL=0
MOVL C01902 V=800.0 PL=0
MOVL C01903 V=800.0 PL=0
MOVL C01904 V=800.0 PL=0
MOVL C01905 V=800.0 PL=0
MOVL C01906 V=800.0 PL=0
MOVL C01907 V=800.0 PL=0
MOVL C01908 V=800.0 PL=0
MOVL C01909 V=800.0 PL=0
MOVL C01910 V=800.0 PL=0
MOVL C01911 V=800.0 PL=0
MOVL C01912 V=800.0 PL=0
MOVL C01913 V=800.0 PL=0
MOVL C01914 V=800.0 PL=0
MOVL C01915 V=800.0 PL=0
MOVL C01916 V=800.0 PL=0
MOVL C01917 V=800.0 PL=0
MOVL C01918 V=800.0 PL=0
MOVL C01919 V=800.0 PL=0
MOVL C01920 V=800.0 PL=0
MOVL C01921 V=800.0 PL=0
MOVL C01922 V=800.0 PL=0
MOVL C01923 V=800.0 PL=0
MOVL C01924 V=800.0 PL=0
MOVL C01925 V=800.0 PL=0
MOVL C01926 V=800.0 PL=0
MOVL C01927 V=800.0 PL=0
MOVL C01928 V=800.0 PL=0
MOVL C01929 V=800.0 PL=0
MOVL C01930 V=800.0 PL=0
MOVL C01931 V=800.0 PL=0
MOVL C01932 V=800.0 PL=0
MOVL C01933 V=800.0 PL=0
MOVL C01934 V=800.0 PL=0
MOVL C01935 V=800.0 PL=0
MOVL C01936 V=800.0 PL=0
MOVL C01937 V=800.0 PL=0
MOVL C01938 V=800.0 PL=0
MOVL C01939 V=800.0 PL=0
MOVL C01940 V=800.0 PL=0
MOVL C01941 V=800.0 PL=0
MOVL C01942 V=800.0 PL=0
MOVL C01943 V=800.0 PL=0
MOVL C01944 V=800.0 PL=0
MOVL C01945 V=800.0 PL=0
MOVL C01946 V=800.0 PL=0
MOVL C01947 V=800.0 PL=0
MOVL C01948 V=800.0 PL=0
MOVL C01949 V=800.0 PL=0
MOVL C01950 V=800.0 PL=0
MOVL C01951 V=800.0 PL=0
MOVL C01952 V=800.0 PL=0
MOVL C01953 V=800.0 PL=0
MOVL C01954 V=800.0 PL=0
MOVL C01955 V=800.0 PL=0
MOVL C01956 V=800.0 PL=0
MOVL C01957 V=800.0 PL=0
MOVL C01958 V=800.0 PL=0
MOVL C01959 V=800.0 PL=0
MOVL C01960 V=800.0 PL=0
MOVL C01961 V=800.0 PL=0
MOVL C01962 V=800.0 PL=0
MOVL C01963 V=800.0 PL=0
MOVL C01964 V=800.0 PL=0
MOVL C01965 V=800.0 PL=0
MOVL C01966 V=800.0 PL=0
MOVL C01967 V=800.0 PL=0
MOVL C01968 V=800.0 PL=0
MOVL C01969 V=800.0 PL=0
MOVL C01970 V=800.0 PL=0
MOVL C01971 V=800.0 PL=0
MOVL C01972 V=800.0 PL=0
MOVL C01973 V=800.0 PL=0
MOVL C01974 V=800.0 PL=0
MOVL C01975 V=800.0 PL=0
MOVL C01976 V=800.0 PL=0
MOVL C01977 V=800.0 PL=0
MOVL C01978 V=800.0 PL=0
MOVL C01979 V=800.0 PL=0
MOVL C01980 V=800.0 PL=0
MOVL C01981 V=800.0 PL=0
MOVL C01982 V=800.0 PL=0
MOVL C01983 V=800.0 PL=0
MOVL C01984 V=800.0 PL=0
MOVL C01985 V=800.0 PL=0
MOVL C01986 V=800.0 PL=0
MOVL C01987 V=800.0 PL=0
MOVL C01988 V=800.0 PL=0
MOVL C01989 V=800.0 PL=0
MOVL C01990 V=800.0 PL=0
MOVL C01991 V=800.0 PL=0
MOVL C01992 V=800.0 PL=0
MOVL C01993 V=800.0 PL=0
MOVL C01994 V=800.0 PL=0
MOVL C01995 V=800.0 PL=0
MOVL C01996 V=800.0 PL=0
MOVL C01997 V=800.0 PL=0
MOVL C01998 V=800.0 PL=0
MOVL C01999 V=800.0 PL=0
MOVL C02000 V=800.0 PL=0
MOVL C02001 V=800.0 PL=0
MOVL C02002 V=800.0 PL=0
MOVL C02003 V=800.0 PL=0
MOVL C02004 V=800.0 PL=0
MOVL C02005 V=800.0 PL=0
MOVL C02006 V=800.0 PL=0
MOVL C02007 V=800.0 PL=0
MOVL C02008 V=800.0 PL=0
MOVL C02009 V=800.0 PL=0
MOVL C02010 V=800.0 PL=0
MOVL C02011 V=800.0 PL=0
MOVL C02012 V=800.0 PL=0
MOVL C02013 V=800.0 PL=0
MOVL C02014 V=800.0 PL=0
MOVL C02015 V=800.0 PL=0
MOVL C02016 V=800.0 PL=0
MOVL C02017 V=800.0 PL=0
MOVL C02018 V=800.0 PL=0
MOVL C02019 V=800.0 PL=0
MOVL C02020 V=800.0 PL=0
MOVL C02021 V=800.0 PL=0
MOVL C02022 V=800.0 PL=0
MOVL C02023 V=800.0 PL=0
MOVL C02024 V=800.0 PL=0
MOVL C02025 V=800.0 PL=0
MOVL C02026 V=800.0 PL=0
MOVL C02027 V=800.0 PL=0
MOVL C02028 V=800.0 PL=0
MOVL C02029 V=800.0 PL=0
MOVL C02030 V=800.0 PL=0
MOVL C02031 V=800.0 PL=0
MOVL C02032 V=800.0 PL=0
MOVL C02033 V=800.0 PL=0
MOVL C02034 V=800.0 PL=0
MOVL C02035 V=800.0 PL=0
MOVL C02036 V=800.0 PL=0
MOVL C02037 V=800.0 PL=0
MOVL C02038 V=800.0 PL=0
MOVL C02039 V=800.0 PL=0
MOVL C02040 V=800.0 PL=0
MOVL C02041 V=800.0 PL=0
MOVL C02042 V=800.0 PL=0
MOVL C02043 V=800.0 PL=0
MOVL C02044 V=800.0 PL=0
MOVL C02045 V=800.0 PL=0
MOVL C02046 V=800.0 PL=0
MOVL C02047 V=800.0 PL=0
MOVL C02048 V=800.0 PL=0
MOVL C02049 V=800.0 PL=0
MOVL C02050 V=800.0 PL=0
MOVL C02051 V=800.0 PL=0
MOVL C02052 V=800.0 PL=0
MOVL C02053 V=800.0 PL=0
MOVL C02054 V=800.0 PL=0
MOVL C02055 V=800.0 PL=0
MOVL C02056 V=800.0 PL=0
MOVL C02057 V=800.0 PL=0
MOVL C02058 V=800.0 PL=0
MOVL C02059 V=800.0 PL=0
MOVL C02060 V=800.0 PL=0
MOVL C02061 V=800.0 PL=0
MOVL C02062 V=800.0 PL=0
MOVL C02063 V=800.0 PL=0
MOVL C02064 V=800.0 PL=0
MOVL C02065 V=800.0 PL=0
MOVL C02066 V=800.0 PL=0
MOVL C02067 V=800.0 PL=0
MOVL C02068 V=800.0 PL=0
MOVL C02069 V=800.0 PL=0
MOVL C02070 V=800.0 PL=0
MOVL C02071 V=800.0 PL=0
MOVL C02072 V=800.0 PL=0
MOVL C02073 V=800.0 PL=0
MOVL C02074 V=800.0 PL=0
MOVL C02075 V=800.0 PL=0
MOVL C02076 V=800.0 PL=0
MOVL C02077 V=800.0 PL=0
MOVL C02078 V=800.0 PL=0
MOVL C02079 V=800.0 PL=0
MOVL C02080 V=800.0 PL=0
